ABB RAPID module: P703.mod

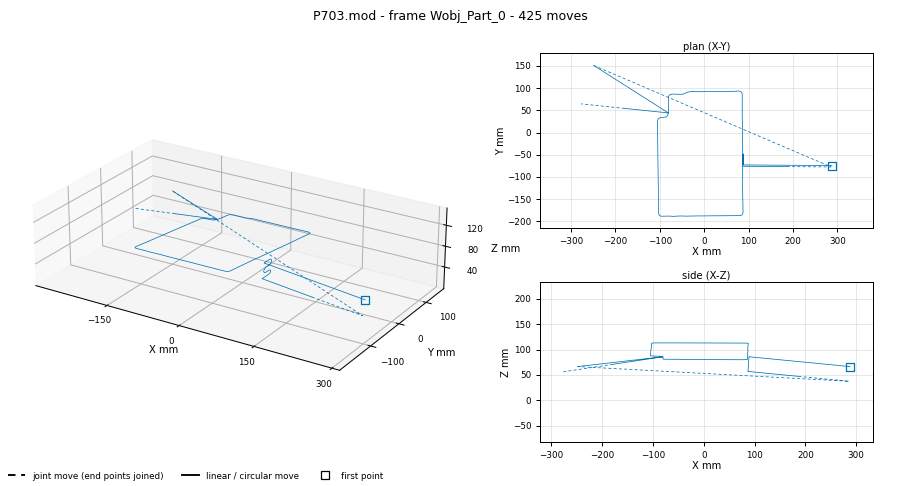
[picture p0: tool path of P703.mod in frame Wobj_Part_0, 425 of 435 moves have a stored position in this frame; points joined in program order, loops and branches not executed]
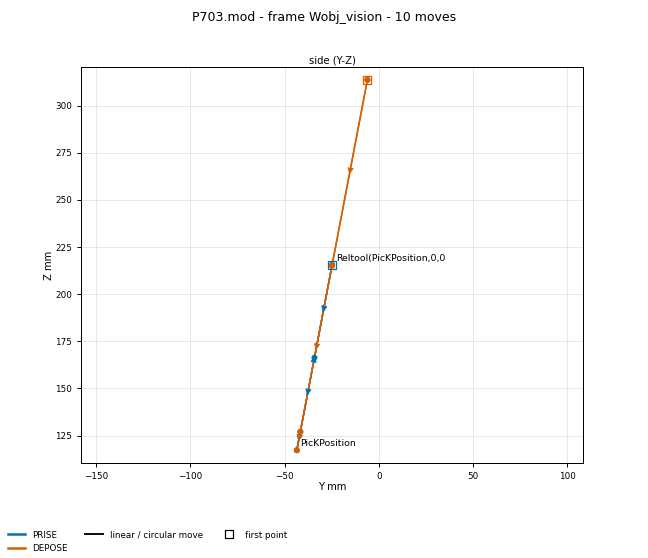
[picture p1: tool path of P703.mod in frame Wobj_vision, 10 of 435 moves have a stored position in this frame; points joined in program order, loops and branches not executed]
MODULE P703

    ! Nom         :P703
    ! Description :
    ! Créé le     :29/05/2023 16:45:30

    LOCAL CONST SPEEDDATA VitesseLente :=[10,500,0,0];
	LOCAL CONST SPEEDDATA VitesseRapide :=[30,500,0,0];
	LOCAL CONST SPEEDDATA VitesseTronconnage :=[2,500,0,0];
	LOCAL CONST SPEEDDATA VitesseTronconnageApp :=[10,500,0,0];
    !
    !Point de prise
    LOCAL PERS Robtarget PicKPosition := [[-18.2045176423154,-43.4890732040902,117.207315713413],[0.0720116404996143,0.704562270319023,0.703344125703762,-0.0609374409822815],[0,0,0,0],[8.999999E+09,8.999999E+09,8.999999E+09,8.999999E+09,8.999999E+09,8.999999E+09]];
	LOCAL PERS Pose Ref := [[0,0,0],[1,0,0,0]];
    !
    !Declaration des points de meulage

    !Tr_meulage_motif_1 : Meulage d'un motif
    LOCAL CONST Robtarget Tr_meulage_motif_1_0 := [[88.8950546875,-72.9881875,85.8599921875],[0.525548833980486,-0.476975326776561,-0.473452006925869,0.521666711498837],[0,0,0,0],[8.999999E+09,8.999999E+09,8.999999E+09,8.999999E+09,8.999999E+09,8.999999E+09]];
    LOCAL CONST Robtarget Tr_meulage_motif_1_1 := [[88.8954296875,-71.9881875,85.8600078125],[0.525548833980486,-0.476975326776561,-0.473452006925869,0.521666711498837],[0,0,0,0],[8.999999E+09,8.999999E+09,8.999999E+09,8.999999E+09,8.999999E+09,8.999999E+09]];
    LOCAL CONST Robtarget Tr_meulage_motif_1_2 := [[88.8958046875,-70.9881875,85.8600234375],[0.525548833980486,-0.476975326776561,-0.473452006925869,0.521666711498837],[0,0,0,0],[8.999999E+09,8.999999E+09,8.999999E+09,8.999999E+09,8.999999E+09,8.999999E+09]];
    LOCAL CONST Robtarget Tr_meulage_motif_1_3 := [[88.8961796875,-69.9881875,85.860046875],[0.525548833980486,-0.476975326776561,-0.473452006925869,0.521666711498837],[0,0,0,0],[8.999999E+09,8.999999E+09,8.999999E+09,8.999999E+09,8.999999E+09,8.999999E+09]];
    LOCAL CONST Robtarget Tr_meulage_motif_1_4 := [[88.8965546875,-68.9881875,85.8600625],[0.525548833980486,-0.476975326776561,-0.473452006925869,0.521666711498837],[0,0,0,0],[8.999999E+09,8.999999E+09,8.999999E+09,8.999999E+09,8.999999E+09,8.999999E+09]];
    LOCAL CONST Robtarget Tr_meulage_motif_1_5 := [[88.8969296875,-67.9881875,85.860078125],[0.525548833980486,-0.476975326776561,-0.473452006925869,0.521666711498837],[0,0,0,0],[8.999999E+09,8.999999E+09,8.999999E+09,8.999999E+09,8.999999E+09,8.999999E+09]];
    LOCAL CONST Robtarget Tr_meulage_motif_1_6 := [[88.8973046875,-66.9881875,85.86009375],[0.525548833980486,-0.476975326776561,-0.473452006925869,0.521666711498837],[0,0,0,0],[8.999999E+09,8.999999E+09,8.999999E+09,8.999999E+09,8.999999E+09,8.999999E+09]];
    LOCAL CONST Robtarget Tr_meulage_motif_1_7 := [[88.897671875,-65.9881875,85.860109375],[0.525548833980486,-0.476975326776561,-0.473452006925869,0.521666711498837],[0,0,0,0],[8.999999E+09,8.999999E+09,8.999999E+09,8.999999E+09,8.999999E+09,8.999999E+09]];
    LOCAL CONST Robtarget Tr_meulage_motif_1_8 := [[88.898046875,-64.98818359375,85.860125],[0.525548833980486,-0.476975326776561,-0.473452006925869,0.521666711498837],[0,0,0,0],[8.999999E+09,8.999999E+09,8.999999E+09,8.999999E+09,8.999999E+09,8.999999E+09]];
    LOCAL CONST Robtarget Tr_meulage_motif_1_9 := [[88.898421875,-63.98818359375,85.8601484375],[0.525548833980486,-0.476975326776561,-0.473452006925869,0.521666711498837],[0,0,0,0],[8.999999E+09,8.999999E+09,8.999999E+09,8.999999E+09,8.999999E+09,8.999999E+09]];
    LOCAL CONST Robtarget Tr_meulage_motif_1_10 := [[88.898796875,-62.98818359375,85.8601640625],[0.525548833980486,-0.476975326776561,-0.473452006925869,0.521666711498837],[0,0,0,0],[8.999999E+09,8.999999E+09,8.999999E+09,8.999999E+09,8.999999E+09,8.999999E+09]];
    LOCAL CONST Robtarget Tr_meulage_motif_1_11 := [[88.899171875,-61.98818359375,85.8601796875],[0.525548833980486,-0.476975326776561,-0.473452006925869,0.521666711498837],[0,0,0,0],[8.999999E+09,8.999999E+09,8.999999E+09,8.999999E+09,8.999999E+09,8.999999E+09]];
    LOCAL CONST Robtarget Tr_meulage_motif_1_12 := [[88.899546875,-60.98818359375,85.8601953125],[0.525548833980486,-0.476975326776561,-0.473452006925869,0.521666711498837],[0,0,0,0],[8.999999E+09,8.999999E+09,8.999999E+09,8.999999E+09,8.999999E+09,8.999999E+09]];
    LOCAL CONST Robtarget Tr_meulage_motif_1_13 := [[88.899921875,-59.98818359375,85.8602109375],[0.525548833980486,-0.476975326776561,-0.473452006925869,0.521666711498837],[0,0,0,0],[8.999999E+09,8.999999E+09,8.999999E+09,8.999999E+09,8.999999E+09,8.999999E+09]];
    LOCAL CONST Robtarget Tr_meulage_motif_1_14 := [[88.900296875,-58.98818359375,85.8602265625],[0.525548833980486,-0.476975326776561,-0.473452006925869,0.521666711498837],[0,0,0,0],[8.999999E+09,8.999999E+09,8.999999E+09,8.999999E+09,8.999999E+09,8.999999E+09]];
    LOCAL CONST Robtarget Tr_meulage_motif_1_15 := [[88.900671875,-57.98818359375,85.8602421875],[0.525548833980486,-0.476975326776561,-0.473452006925869,0.521666711498837],[0,0,0,0],[8.999999E+09,8.999999E+09,8.999999E+09,8.999999E+09,8.999999E+09,8.999999E+09]];
    LOCAL CONST Robtarget Tr_meulage_motif_1_16 := [[88.901046875,-56.98818359375,85.860265625],[0.525548833980486,-0.476975326776561,-0.473452006925869,0.521666711498837],[0,0,0,0],[8.999999E+09,8.999999E+09,8.999999E+09,8.999999E+09,8.999999E+09,8.999999E+09]];
    LOCAL CONST Robtarget Tr_meulage_motif_1_17 := [[88.901421875,-55.98818359375,85.86028125],[0.525548833980486,-0.476975326776561,-0.473452006925869,0.521666711498837],[0,0,0,0],[8.999999E+09,8.999999E+09,8.999999E+09,8.999999E+09,8.999999E+09,8.999999E+09]];
    LOCAL CONST Robtarget Tr_meulage_motif_1_18 := [[88.901796875,-54.98818359375,85.860296875],[0.525548833980486,-0.476975326776561,-0.473452006925869,0.521666711498837],[0,0,0,0],[8.999999E+09,8.999999E+09,8.999999E+09,8.999999E+09,8.999999E+09,8.999999E+09]];
    LOCAL CONST Robtarget Tr_meulage_motif_1_19 := [[88.8946171875,-53.9956171875,85.7499765625],[0.525548833980486,-0.476975326776561,-0.473452006925869,0.521666711498837],[0,0,0,0],[8.999999E+09,8.999999E+09,8.999999E+09,8.999999E+09,8.999999E+09,8.999999E+09]];
    LOCAL CONST Robtarget Tr_meulage_motif_1_20 := [[88.8805546875,-53.049109375,85.539296875],[0.525548833980486,-0.476975326776561,-0.473452006925869,0.521666711498837],[0,0,0,0],[8.999999E+09,8.999999E+09,8.999999E+09,8.999999E+09,8.999999E+09,8.999999E+09]];
    LOCAL CONST Robtarget Tr_meulage_motif_1_21 := [[88.8623203125,-52.19637890625,85.2681015625],[0.525548833980486,-0.476975326776561,-0.473452006925869,0.521666711498837],[0,0,0,0],[8.999999E+09,8.999999E+09,8.999999E+09,8.999999E+09,8.999999E+09,8.999999E+09]];
    LOCAL CONST Robtarget Tr_meulage_motif_1_22 := [[88.843765625,-51.4464296875,84.9928203125],[0.525548833980486,-0.476975326776561,-0.473452006925869,0.521666711498837],[0,0,0,0],[8.999999E+09,8.999999E+09,8.999999E+09,8.999999E+09,8.999999E+09,8.999999E+09]];
    LOCAL CONST Robtarget Tr_meulage_motif_1_23 := [[88.8021171875,-50.34533984375,84.3781484375],[0.525548833980486,-0.476975326776561,-0.473452006925869,0.521666711498837],[0,0,0,0],[8.999999E+09,8.999999E+09,8.999999E+09,8.999999E+09,8.999999E+09,8.999999E+09]];
    LOCAL CONST Robtarget Tr_meulage_motif_1_24 := [[88.744640625,-49.3214296875,83.5324921875],[0.525548833980486,-0.476975326776561,-0.473452006925869,0.521666711498837],[0,0,0,0],[8.999999E+09,8.999999E+09,8.999999E+09,8.999999E+09,8.999999E+09,8.999999E+09]];
    LOCAL CONST Robtarget Tr_meulage_motif_1_25 := [[88.6750625,-48.47373046875,82.511015625],[0.525548833980486,-0.476975326776561,-0.473452006925869,0.521666711498837],[0,0,0,0],[8.999999E+09,8.999999E+09,8.999999E+09,8.999999E+09,8.999999E+09,8.999999E+09]];
    LOCAL CONST Robtarget Tr_meulage_motif_1_26 := [[88.5990546875,-47.98552734375,81.3974453125],[0.525548833980486,-0.476975326776561,-0.473452006925869,0.521666711498837],[0,0,0,0],[8.999999E+09,8.999999E+09,8.999999E+09,8.999999E+09,8.999999E+09,8.999999E+09]];
    LOCAL CONST Robtarget Tr_meulage_motif_1_27 := [[88.5515546875,-47.95843359375,80.70309375],[0.525548833980486,-0.476975326776561,-0.473452006925869,0.521666711498837],[0,0,0,0],[8.999999E+09,8.999999E+09,8.999999E+09,8.999999E+09,8.999999E+09,8.999999E+09]];
    LOCAL CONST Robtarget Tr_meulage_motif_1_28 := [[88.506421875,-47.95840625,80.043390625],[0.525548833980486,-0.476975326776561,-0.473452006925869,0.521666711498837],[0,0,0,0],[8.999999E+09,8.999999E+09,8.999999E+09,8.999999E+09,8.999999E+09,8.999999E+09]];
    LOCAL CONST Robtarget Tr_meulage_motif_1_29 := [[88.4612734375,-48.01325390625,79.3838359375],[0.525548833980486,-0.476975326776561,-0.473452006925869,0.521666711498837],[0,0,0,0],[8.999999E+09,8.999999E+09,8.999999E+09,8.999999E+09,8.999999E+09,8.999999E+09]];
    LOCAL CONST Robtarget Tr_meulage_motif_1_30 := [[88.385875,-48.51142578125,78.2846484375],[0.525548833980486,-0.476975326776561,-0.473452006925869,0.521666711498837],[0,0,0,0],[8.999999E+09,8.999999E+09,8.999999E+09,8.999999E+09,8.999999E+09,8.999999E+09]];
    LOCAL CONST Robtarget Tr_meulage_motif_1_31 := [[88.31684375,-49.3680078125,77.280359375],[0.525548833980486,-0.476975326776561,-0.473452006925869,0.521666711498837],[0,0,0,0],[8.999999E+09,8.999999E+09,8.999999E+09,8.999999E+09,8.999999E+09,8.999999E+09]];
    LOCAL CONST Robtarget Tr_meulage_motif_1_32 := [[88.2598828125,-50.39137890625,76.4533984375],[0.525548833980486,-0.476975326776561,-0.473452006925869,0.521666711498837],[0,0,0,0],[8.999999E+09,8.999999E+09,8.999999E+09,8.999999E+09,8.999999E+09,8.999999E+09]];
    LOCAL CONST Robtarget Tr_meulage_motif_1_33 := [[88.232609375,-51.07845703125,76.0585625],[0.525548833980486,-0.476975326776561,-0.473452006925869,0.521666711498837],[0,0,0,0],[8.999999E+09,8.999999E+09,8.999999E+09,8.999999E+09,8.999999E+09,8.999999E+09]];
    LOCAL CONST Robtarget Tr_meulage_motif_1_34 := [[88.1988984375,-52.23659375,75.5721484375],[0.525548833980486,-0.476975326776561,-0.473452006925869,0.521666711498837],[0,0,0,0],[8.999999E+09,8.999999E+09,8.999999E+09,8.999999E+09,8.999999E+09,8.999999E+09]];
    LOCAL CONST Robtarget Tr_meulage_motif_1_35 := [[88.1805546875,-53.08161328125,75.30865625],[0.525548833980486,-0.476975326776561,-0.473452006925869,0.521666711498837],[0,0,0,0],[8.999999E+09,8.999999E+09,8.999999E+09,8.999999E+09,8.999999E+09,8.999999E+09]];
    LOCAL CONST Robtarget Tr_meulage_motif_1_36 := [[88.16625,-54.0136015625,75.1046484375],[0.525548833980486,-0.476975326776561,-0.473452006925869,0.521666711498837],[0,0,0,0],[8.999999E+09,8.999999E+09,8.999999E+09,8.999999E+09,8.999999E+09,8.999999E+09]];
    LOCAL CONST Robtarget Tr_meulage_motif_1_37 := [[88.15846875,-54.99516015625,74.9962890625],[0.525548833980486,-0.476975326776561,-0.473452006925869,0.521666711498837],[0,0,0,0],[8.999999E+09,8.999999E+09,8.999999E+09,8.999999E+09,8.999999E+09,8.999999E+09]];
    LOCAL CONST Robtarget Tr_meulage_motif_1_38 := [[88.150546875,-55.98771875,74.8859375],[0.525548833980486,-0.476975326776561,-0.473452006925869,0.521666711498837],[0,0,0,0],[8.999999E+09,8.999999E+09,8.999999E+09,8.999999E+09,8.999999E+09,8.999999E+09]];
    LOCAL CONST Robtarget Tr_meulage_motif_1_39 := [[88.150171875,-56.98771875,74.885921875],[0.525548833980486,-0.476975326776561,-0.473452006925869,0.521666711498837],[0,0,0,0],[8.999999E+09,8.999999E+09,8.999999E+09,8.999999E+09,8.999999E+09,8.999999E+09]];
    LOCAL CONST Robtarget Tr_meulage_motif_1_40 := [[88.149796875,-57.98771875,74.88590625],[0.525548833980486,-0.476975326776561,-0.473452006925869,0.521666711498837],[0,0,0,0],[8.999999E+09,8.999999E+09,8.999999E+09,8.999999E+09,8.999999E+09,8.999999E+09]];
    LOCAL CONST Robtarget Tr_meulage_motif_1_41 := [[88.149421875,-58.98771875,74.8858828125],[0.525548833980486,-0.476975326776561,-0.473452006925869,0.521666711498837],[0,0,0,0],[8.999999E+09,8.999999E+09,8.999999E+09,8.999999E+09,8.999999E+09,8.999999E+09]];
    LOCAL CONST Robtarget Tr_meulage_motif_1_42 := [[88.149046875,-59.98771875,74.8858671875],[0.525548833980486,-0.476975326776561,-0.473452006925869,0.521666711498837],[0,0,0,0],[8.999999E+09,8.999999E+09,8.999999E+09,8.999999E+09,8.999999E+09,8.999999E+09]];
    LOCAL CONST Robtarget Tr_meulage_motif_1_43 := [[88.148671875,-60.98771875,74.8858515625],[0.525548833980486,-0.476975326776561,-0.473452006925869,0.521666711498837],[0,0,0,0],[8.999999E+09,8.999999E+09,8.999999E+09,8.999999E+09,8.999999E+09,8.999999E+09]];
    LOCAL CONST Robtarget Tr_meulage_motif_1_44 := [[88.148296875,-61.98771875,74.8858359375],[0.525548833980486,-0.476975326776561,-0.473452006925869,0.521666711498837],[0,0,0,0],[8.999999E+09,8.999999E+09,8.999999E+09,8.999999E+09,8.999999E+09,8.999999E+09]];
    LOCAL CONST Robtarget Tr_meulage_motif_1_45 := [[88.147921875,-62.98771875,74.8858203125],[0.525548833980486,-0.476975326776561,-0.473452006925869,0.521666711498837],[0,0,0,0],[8.999999E+09,8.999999E+09,8.999999E+09,8.999999E+09,8.999999E+09,8.999999E+09]];
    LOCAL CONST Robtarget Tr_meulage_motif_1_46 := [[88.147546875,-63.98771875,74.8858046875],[0.525548833980486,-0.476975326776561,-0.473452006925869,0.521666711498837],[0,0,0,0],[8.999999E+09,8.999999E+09,8.999999E+09,8.999999E+09,8.999999E+09,8.999999E+09]];
    LOCAL CONST Robtarget Tr_meulage_motif_1_47 := [[88.1471796875,-64.98771875,74.8857890625],[0.525548833980486,-0.476975326776561,-0.473452006925869,0.521666711498837],[0,0,0,0],[8.999999E+09,8.999999E+09,8.999999E+09,8.999999E+09,8.999999E+09,8.999999E+09]];
    LOCAL CONST Robtarget Tr_meulage_motif_1_48 := [[88.1468046875,-65.98771875,74.885765625],[0.525548833980486,-0.476975326776561,-0.473452006925869,0.521666711498837],[0,0,0,0],[8.999999E+09,8.999999E+09,8.999999E+09,8.999999E+09,8.999999E+09,8.999999E+09]];
    LOCAL CONST Robtarget Tr_meulage_motif_1_49 := [[88.1388828125,-66.9802734375,74.7754140625],[0.525548833980486,-0.476975326776561,-0.473452006925869,0.521666711498837],[0,0,0,0],[8.999999E+09,8.999999E+09,8.999999E+09,8.999999E+09,8.999999E+09,8.999999E+09]];
    LOCAL CONST Robtarget Tr_meulage_motif_1_50 := [[88.124109375,-67.926765625,74.564703125],[0.525548833980486,-0.476975326776561,-0.473452006925869,0.521666711498837],[0,0,0,0],[8.999999E+09,8.999999E+09,8.999999E+09,8.999999E+09,8.999999E+09,8.999999E+09]];
    LOCAL CONST Robtarget Tr_meulage_motif_1_51 := [[88.105234375,-68.7794765625,74.293484375],[0.525548833980486,-0.476975326776561,-0.473452006925869,0.521666711498837],[0,0,0,0],[8.999999E+09,8.999999E+09,8.999999E+09,8.999999E+09,8.999999E+09,8.999999E+09]];
    LOCAL CONST Robtarget Tr_meulage_motif_1_52 := [[88.084203125,-69.4909609375,73.9900234375],[0.525548833980486,-0.476975326776561,-0.473452006925869,0.521666711498837],[0,0,0,0],[8.999999E+09,8.999999E+09,8.999999E+09,8.999999E+09,8.999999E+09,8.999999E+09]];
    LOCAL CONST Robtarget Tr_meulage_motif_1_53 := [[88.03859375,-70.5253984375,73.329015625],[0.525548833980486,-0.476975326776561,-0.473452006925869,0.521666711498837],[0,0,0,0],[8.999999E+09,8.999999E+09,8.999999E+09,8.999999E+09,8.999999E+09,8.999999E+09]];
    LOCAL CONST Robtarget Tr_meulage_motif_1_54 := [[87.9766875,-71.4273046875,72.429171875],[0.525548833980486,-0.476975326776561,-0.473452006925869,0.521666711498837],[0,0,0,0],[8.999999E+09,8.999999E+09,8.999999E+09,8.999999E+09,8.999999E+09,8.999999E+09]];
    LOCAL CONST Robtarget Tr_meulage_motif_1_55 := [[87.9050859375,-71.9622265625,71.3855703125],[0.525548833980486,-0.476975326776561,-0.473452006925869,0.521666711498837],[0,0,0,0],[8.999999E+09,8.999999E+09,8.999999E+09,8.999999E+09,8.999999E+09,8.999999E+09]];
    LOCAL CONST Robtarget Tr_meulage_motif_1_56 := [[87.8576953125,-72.1469765625,70.6939609375],[0.525548833980486,-0.476975326776561,-0.473452006925869,0.521666711498837],[0,0,0,0],[8.999999E+09,8.999999E+09,8.999999E+09,8.999999E+09,8.999999E+09,8.999999E+09]];
    LOCAL CONST Robtarget Tr_meulage_motif_1_57 := [[87.805109375,-72.2107890625,69.9257578125],[0.525548833980486,-0.476975326776561,-0.473452006925869,0.521666711498837],[0,0,0,0],[8.999999E+09,8.999999E+09,8.999999E+09,8.999999E+09,8.999999E+09,8.999999E+09]];
    LOCAL CONST Robtarget Tr_meulage_motif_1_58 := [[87.7525859375,-72.1438203125,69.1576796875],[0.525548833980486,-0.476975326776561,-0.473452006925869,0.521666711498837],[0,0,0,0],[8.999999E+09,8.999999E+09,8.999999E+09,8.999999E+09,8.999999E+09,8.999999E+09]];
    LOCAL CONST Robtarget Tr_meulage_motif_1_59 := [[87.67709375,-71.7241796875,68.0520234375],[0.525548833980486,-0.476975326776561,-0.473452006925869,0.521666711498837],[0,0,0,0],[8.999999E+09,8.999999E+09,8.999999E+09,8.999999E+09,8.999999E+09,8.999999E+09]];
    LOCAL CONST Robtarget Tr_meulage_motif_1_60 := [[87.637265625,-71.30984375,67.4677109375],[0.525548833980486,-0.476975326776561,-0.473452006925869,0.521666711498837],[0,0,0,0],[8.999999E+09,8.999999E+09,8.999999E+09,8.999999E+09,8.999999E+09,8.999999E+09]];
    LOCAL CONST Robtarget Tr_meulage_motif_1_61 := [[87.5770390625,-70.4226796875,66.582671875],[0.525548833980486,-0.476975326776561,-0.473452006925869,0.521666711498837],[0,0,0,0],[8.999999E+09,8.999999E+09,8.999999E+09,8.999999E+09,8.999999E+09,8.999999E+09]];
    LOCAL CONST Robtarget Tr_meulage_motif_1_62 := [[87.5489765625,-69.8369765625,66.1693359375],[0.525548833980486,-0.476975326776561,-0.473452006925869,0.521666711498837],[0,0,0,0],[8.999999E+09,8.999999E+09,8.999999E+09,8.999999E+09,8.999999E+09,8.999999E+09]];
    LOCAL CONST Robtarget Tr_meulage_motif_1_63 := [[87.5122578125,-68.719046875,65.6265234375],[0.525548833980486,-0.476975326776561,-0.473452006925869,0.521666711498837],[0,0,0,0],[8.999999E+09,8.999999E+09,8.999999E+09,8.999999E+09,8.999999E+09,8.999999E+09]];
    LOCAL CONST Robtarget Tr_meulage_motif_1_64 := [[87.4923984375,-67.8934375,65.33173046875],[0.525548833980486,-0.476975326776561,-0.473452006925869,0.521666711498837],[0,0,0,0],[8.999999E+09,8.999999E+09,8.999999E+09,8.999999E+09,8.999999E+09,8.999999E+09]];
    LOCAL CONST Robtarget Tr_meulage_motif_1_65 := [[87.4787890625,-66.9614296875,65.12775390625],[0.525548833980486,-0.476975326776561,-0.473452006925869,0.521666711498837],[0,0,0,0],[8.999999E+09,8.999999E+09,8.999999E+09,8.999999E+09,8.999999E+09,8.999999E+09]];
    LOCAL CONST Robtarget Tr_meulage_motif_1_66 := [[87.4717421875,-65.979859375,65.0194296875],[0.525548833980486,-0.476975326776561,-0.473452006925869,0.521666711498837],[0,0,0,0],[8.999999E+09,8.999999E+09,8.999999E+09,8.999999E+09,8.999999E+09,8.999999E+09]];
    LOCAL CONST Robtarget Tr_meulage_motif_1_67 := [[87.4645625,-64.98729296875,64.909109375],[0.525548833980486,-0.476975326776561,-0.473452006925869,0.521666711498837],[0,0,0,0],[8.999999E+09,8.999999E+09,8.999999E+09,8.999999E+09,8.999999E+09,8.999999E+09]];
    LOCAL CONST Robtarget Tr_meulage_motif_1_68 := [[87.4649375,-63.98729296875,64.90912890625],[0.525548833980486,-0.476975326776561,-0.473452006925869,0.521666711498837],[0,0,0,0],[8.999999E+09,8.999999E+09,8.999999E+09,8.999999E+09,8.999999E+09,8.999999E+09]];
    LOCAL CONST Robtarget Tr_meulage_motif_1_69 := [[87.4653125,-62.98729296875,64.90914453125],[0.525548833980486,-0.476975326776561,-0.473452006925869,0.521666711498837],[0,0,0,0],[8.999999E+09,8.999999E+09,8.999999E+09,8.999999E+09,8.999999E+09,8.999999E+09]];
    LOCAL CONST Robtarget Tr_meulage_motif_1_70 := [[87.4656875,-61.987296875,64.90916015625],[0.525548833980486,-0.476975326776561,-0.473452006925869,0.521666711498837],[0,0,0,0],[8.999999E+09,8.999999E+09,8.999999E+09,8.999999E+09,8.999999E+09,8.999999E+09]];
    LOCAL CONST Robtarget Tr_meulage_motif_1_71 := [[87.4660625,-60.987296875,64.9091796875],[0.525548833980486,-0.476975326776561,-0.473452006925869,0.521666711498837],[0,0,0,0],[8.999999E+09,8.999999E+09,8.999999E+09,8.999999E+09,8.999999E+09,8.999999E+09]];
    LOCAL CONST Robtarget Tr_meulage_motif_1_72 := [[87.4664375,-59.987296875,64.9091953125],[0.525548833980486,-0.476975326776561,-0.473452006925869,0.521666711498837],[0,0,0,0],[8.999999E+09,8.999999E+09,8.999999E+09,8.999999E+09,8.999999E+09,8.999999E+09]];
    LOCAL CONST Robtarget Tr_meulage_motif_1_73 := [[87.4668125,-58.987296875,64.9092109375],[0.525548833980486,-0.476975326776561,-0.473452006925869,0.521666711498837],[0,0,0,0],[8.999999E+09,8.999999E+09,8.999999E+09,8.999999E+09,8.999999E+09,8.999999E+09]];
    LOCAL CONST Robtarget Tr_meulage_motif_1_74 := [[87.4671875,-57.987296875,64.90923046875],[0.525548833980486,-0.476975326776561,-0.473452006925869,0.521666711498837],[0,0,0,0],[8.999999E+09,8.999999E+09,8.999999E+09,8.999999E+09,8.999999E+09,8.999999E+09]];
    LOCAL CONST Robtarget Tr_meulage_motif_1_75 := [[87.4675625,-56.987296875,64.90924609375],[0.525548833980486,-0.476975326776561,-0.473452006925869,0.521666711498837],[0,0,0,0],[8.999999E+09,8.999999E+09,8.999999E+09,8.999999E+09,8.999999E+09,8.999999E+09]];
    LOCAL CONST Robtarget Tr_meulage_motif_1_76 := [[87.4679296875,-55.987296875,64.90926171875],[0.525548833980486,-0.476975326776561,-0.473452006925869,0.521666711498837],[0,0,0,0],[8.999999E+09,8.999999E+09,8.999999E+09,8.999999E+09,8.999999E+09,8.999999E+09]];
    LOCAL CONST Robtarget Tr_meulage_motif_1_77 := [[87.4683046875,-54.987296875,64.90927734375],[0.525548833980486,-0.476975326776561,-0.473452006925869,0.521666711498837],[0,0,0,0],[8.999999E+09,8.999999E+09,8.999999E+09,8.999999E+09,8.999999E+09,8.999999E+09]];
    LOCAL CONST Robtarget Tr_meulage_motif_1_78 := [[87.4611328125,-53.9947265625,64.7989609375],[0.525548833980486,-0.476975326776561,-0.473452006925869,0.521666711498837],[0,0,0,0],[8.999999E+09,8.999999E+09,8.999999E+09,8.999999E+09,8.999999E+09,8.999999E+09]];
    LOCAL CONST Robtarget Tr_meulage_motif_1_79 := [[87.4470703125,-53.04821875,64.58828125],[0.525548833980486,-0.476975326776561,-0.473452006925869,0.521666711498837],[0,0,0,0],[8.999999E+09,8.999999E+09,8.999999E+09,8.999999E+09,8.999999E+09,8.999999E+09]];
    LOCAL CONST Robtarget Tr_meulage_motif_1_80 := [[87.428828125,-52.19548828125,64.3170859375],[0.525548833980486,-0.476975326776561,-0.473452006925869,0.521666711498837],[0,0,0,0],[8.999999E+09,8.999999E+09,8.999999E+09,8.999999E+09,8.999999E+09,8.999999E+09]];
    LOCAL CONST Robtarget Tr_meulage_motif_1_81 := [[87.4102734375,-51.4455390625,64.0418046875],[0.525548833980486,-0.476975326776561,-0.473452006925869,0.521666711498837],[0,0,0,0],[8.999999E+09,8.999999E+09,8.999999E+09,8.999999E+09,8.999999E+09,8.999999E+09]];
    LOCAL CONST Robtarget Tr_meulage_motif_1_82 := [[87.3686328125,-50.344453125,63.42713671875],[0.525548833980486,-0.476975326776561,-0.473452006925869,0.521666711498837],[0,0,0,0],[8.999999E+09,8.999999E+09,8.999999E+09,8.999999E+09,8.999999E+09,8.999999E+09]];
    LOCAL CONST Robtarget Tr_meulage_motif_1_83 := [[87.30796875,-49.3876953125,62.53526953125],[0.525548833980486,-0.476975326776561,-0.473452006925869,0.521666711498837],[0,0,0,0],[8.999999E+09,8.999999E+09,8.999999E+09,8.999999E+09,8.999999E+09,8.999999E+09]];
    LOCAL CONST Robtarget Tr_meulage_motif_1_84 := [[87.2340625,-48.7785234375,61.4518125],[0.525548833980486,-0.476975326776561,-0.473452006925869,0.521666711498837],[0,0,0,0],[8.999999E+09,8.999999E+09,8.999999E+09,8.999999E+09,8.999999E+09,8.999999E+09]];
    LOCAL CONST Robtarget Tr_meulage_motif_1_85 := [[87.1669296875,-48.60916796875,60.469734375],[0.525548833980486,-0.476975326776561,-0.473452006925869,0.521666711498837],[0,0,0,0],[8.999999E+09,8.999999E+09,8.999999E+09,8.999999E+09,8.999999E+09,8.999999E+09]];
    LOCAL CONST Robtarget Tr_meulage_motif_1_86 := [[87.1529140625,-48.74062890625,60.2655546875],[0.525548833980486,-0.476975326776561,-0.473452006925869,0.521666711498837],[0,0,0,0],[8.999999E+09,8.999999E+09,8.999999E+09,8.999999E+09,8.999999E+09,8.999999E+09]];
    LOCAL CONST Robtarget Tr_meulage_motif_1_87 := [[87.10328125,-48.86397265625,59.54083984375],[0.525548833980486,-0.476975326776561,-0.473452006925869,0.521666711498837],[0,0,0,0],[8.999999E+09,8.999999E+09,8.999999E+09,8.999999E+09,8.999999E+09,8.999999E+09]];
    LOCAL CONST Robtarget Tr_meulage_motif_1_88 := [[87.0390703125,-49.54793359375,58.606109375],[0.525548833980486,-0.476975326776561,-0.473452006925869,0.521666711498837],[0,0,0,0],[8.999999E+09,8.999999E+09,8.999999E+09,8.999999E+09,8.999999E+09,8.999999E+09]];
    LOCAL CONST Robtarget Tr_meulage_motif_1_89 := [[87.007203125,-50.1055390625,58.1433671875],[0.525548833980486,-0.476975326776561,-0.473452006925869,0.521666711498837],[0,0,0,0],[8.999999E+09,8.999999E+09,8.999999E+09,8.999999E+09,8.999999E+09,8.999999E+09]];
    LOCAL CONST Robtarget Tr_meulage_motif_1_90 := [[86.9705703125,-51.235828125,57.6141484375],[0.525548833980486,-0.476975326776561,-0.473452006925869,0.521666711498837],[0,0,0,0],[8.999999E+09,8.999999E+09,8.999999E+09,8.999999E+09,8.999999E+09,8.999999E+09]];
    LOCAL CONST Robtarget Tr_meulage_motif_1_91 := [[86.9522265625,-52.0808515625,57.35065625],[0.525548833980486,-0.476975326776561,-0.473452006925869,0.521666711498837],[0,0,0,0],[8.999999E+09,8.999999E+09,8.999999E+09,8.999999E+09,8.999999E+09,8.999999E+09]];
    LOCAL CONST Robtarget Tr_meulage_motif_1_92 := [[86.937921875,-53.01283984375,57.1466484375],[0.525548833980486,-0.476975326776561,-0.473452006925869,0.521666711498837],[0,0,0,0],[8.999999E+09,8.999999E+09,8.999999E+09,8.999999E+09,8.999999E+09,8.999999E+09]];
    LOCAL CONST Robtarget Tr_meulage_motif_1_93 := [[86.930140625,-53.9943984375,57.03829296875],[0.525548833980486,-0.476975326776561,-0.473452006925869,0.521666711498837],[0,0,0,0],[8.999999E+09,8.999999E+09,8.999999E+09,8.999999E+09,8.999999E+09,8.999999E+09]];
    LOCAL CONST Robtarget Tr_meulage_motif_1_94 := [[86.92221875,-54.98695703125,56.9279375],[0.525548833980486,-0.476975326776561,-0.473452006925869,0.521666711498837],[0,0,0,0],[8.999999E+09,8.999999E+09,8.999999E+09,8.999999E+09,8.999999E+09,8.999999E+09]];
    LOCAL CONST Robtarget Tr_meulage_motif_1_95 := [[86.92184375,-55.98695703125,56.927921875],[0.525548833980486,-0.476975326776561,-0.473452006925869,0.521666711498837],[0,0,0,0],[8.999999E+09,8.999999E+09,8.999999E+09,8.999999E+09,8.999999E+09,8.999999E+09]];
    LOCAL CONST Robtarget Tr_meulage_motif_1_96 := [[86.92146875,-56.98695703125,56.92790625],[0.525548833980486,-0.476975326776561,-0.473452006925869,0.521666711498837],[0,0,0,0],[8.999999E+09,8.999999E+09,8.999999E+09,8.999999E+09,8.999999E+09,8.999999E+09]];
    LOCAL CONST Robtarget Tr_meulage_motif_1_97 := [[86.92109375,-57.98695703125,56.92788671875],[0.525548833980486,-0.476975326776561,-0.473452006925869,0.521666711498837],[0,0,0,0],[8.999999E+09,8.999999E+09,8.999999E+09,8.999999E+09,8.999999E+09,8.999999E+09]];
    LOCAL CONST Robtarget Tr_meulage_motif_1_98 := [[86.92071875,-58.98695703125,56.92787109375],[0.525548833980486,-0.476975326776561,-0.473452006925869,0.521666711498837],[0,0,0,0],[8.999999E+09,8.999999E+09,8.999999E+09,8.999999E+09,8.999999E+09,8.999999E+09]];
    LOCAL CONST Robtarget Tr_meulage_motif_1_99 := [[86.92034375,-59.98695703125,56.92785546875],[0.525548833980486,-0.476975326776561,-0.473452006925869,0.521666711498837],[0,0,0,0],[8.999999E+09,8.999999E+09,8.999999E+09,8.999999E+09,8.999999E+09,8.999999E+09]];
    LOCAL CONST Robtarget Tr_meulage_motif_1_100 := [[86.91996875,-60.98695703125,56.92783984375],[0.525548833980486,-0.476975326776561,-0.473452006925869,0.521666711498837],[0,0,0,0],[8.999999E+09,8.999999E+09,8.999999E+09,8.999999E+09,8.999999E+09,8.999999E+09]];
    LOCAL CONST Robtarget Tr_meulage_motif_1_101 := [[86.91959375,-61.98695703125,56.9278203125],[0.525548833980486,-0.476975326776561,-0.473452006925869,0.521666711498837],[0,0,0,0],[8.999999E+09,8.999999E+09,8.999999E+09,8.999999E+09,8.999999E+09,8.999999E+09]];
    LOCAL CONST Robtarget Tr_meulage_motif_1_102 := [[86.9192265625,-62.98695703125,56.9278046875],[0.525548833980486,-0.476975326776561,-0.473452006925869,0.521666711498837],[0,0,0,0],[8.999999E+09,8.999999E+09,8.999999E+09,8.999999E+09,8.999999E+09,8.999999E+09]];
    LOCAL CONST Robtarget Tr_meulage_motif_1_103 := [[86.9188515625,-63.98695703125,56.9277890625],[0.525548833980486,-0.476975326776561,-0.473452006925869,0.521666711498837],[0,0,0,0],[8.999999E+09,8.999999E+09,8.999999E+09,8.999999E+09,8.999999E+09,8.999999E+09]];
    LOCAL CONST Robtarget Tr_meulage_motif_1_104 := [[86.9184765625,-64.98695703125,56.92776953125],[0.525548833980486,-0.476975326776561,-0.473452006925869,0.521666711498837],[0,0,0,0],[8.999999E+09,8.999999E+09,8.999999E+09,8.999999E+09,8.999999E+09,8.999999E+09]];
    LOCAL CONST Robtarget Tr_meulage_motif_1_105 := [[86.9181015625,-65.986953125,56.92775390625],[0.525548833980486,-0.476975326776561,-0.473452006925869,0.521666711498837],[0,0,0,0],[8.999999E+09,8.999999E+09,8.999999E+09,8.999999E+09,8.999999E+09,8.999999E+09]];
    LOCAL CONST Robtarget Tr_meulage_motif_1_106 := [[86.9177265625,-66.986953125,56.92773828125],[0.525548833980486,-0.476975326776561,-0.473452006925869,0.521666711498837],[0,0,0,0],[8.999999E+09,8.999999E+09,8.999999E+09,8.999999E+09,8.999999E+09,8.999999E+09]];
    LOCAL CONST Robtarget Tr_meulage_motif_1_107 := [[86.9173515625,-67.986953125,56.92771875],[0.525548833980486,-0.476975326776561,-0.473452006925869,0.521666711498837],[0,0,0,0],[8.999999E+09,8.999999E+09,8.999999E+09,8.999999E+09,8.999999E+09,8.999999E+09]];
    LOCAL CONST Robtarget Tr_meulage_motif_1_108 := [[86.9169765625,-68.986953125,56.927703125],[0.525548833980486,-0.476975326776561,-0.473452006925869,0.521666711498837],[0,0,0,0],[8.999999E+09,8.999999E+09,8.999999E+09,8.999999E+09,8.999999E+09,8.999999E+09]];
    LOCAL CONST Robtarget Tr_meulage_motif_1_109 := [[86.9166015625,-69.986953125,56.9276875],[0.525548833980486,-0.476975326776561,-0.473452006925869,0.521666711498837],[0,0,0,0],[8.999999E+09,8.999999E+09,8.999999E+09,8.999999E+09,8.999999E+09,8.999999E+09]];
    LOCAL CONST Robtarget Tr_meulage_motif_1_110 := [[86.9162265625,-70.986953125,56.92766796875],[0.525548833980486,-0.476975326776561,-0.473452006925869,0.521666711498837],[0,0,0,0],[8.999999E+09,8.999999E+09,8.999999E+09,8.999999E+09,8.999999E+09,8.999999E+09]];
    LOCAL CONST Robtarget Tr_meulage_motif_1_111 := [[86.9158515625,-71.986953125,56.92765234375],[0.525548833980486,-0.476975326776561,-0.473452006925869,0.521666711498837],[0,0,0,0],[8.999999E+09,8.999999E+09,8.999999E+09,8.999999E+09,8.999999E+09,8.999999E+09]];
    LOCAL CONST Robtarget Tr_meulage_motif_1_112 := [[86.9154765625,-72.986953125,56.92763671875],[0.525548833980486,-0.476975326776561,-0.473452006925869,0.521666711498837],[0,0,0,0],[8.999999E+09,8.999999E+09,8.999999E+09,8.999999E+09,8.999999E+09,8.999999E+09]];
    LOCAL CONST Robtarget Tr_meulage_motif_1_113 := [[86.9151015625,-73.986953125,56.9276171875],[0.525548833980486,-0.476975326776561,-0.473452006925869,0.521666711498837],[0,0,0,0],[8.999999E+09,8.999999E+09,8.999999E+09,8.999999E+09,8.999999E+09,8.999999E+09]];
    LOCAL CONST Robtarget Tr_meulage_motif_1_114 := [[86.914734375,-74.986953125,56.9276015625],[0.525548833980486,-0.476975326776561,-0.473452006925869,0.521666711498837],[0,0,0,0],[8.999999E+09,8.999999E+09,8.999999E+09,8.999999E+09,8.999999E+09,8.999999E+09]];
    LOCAL CONST Robtarget Tr_meulage_motif_1_115 := [[86.914359375,-75.986953125,56.9275859375],[0.525548833980486,-0.476975326776561,-0.473452006925869,0.521666711498837],[0,0,0,0],[8.999999E+09,8.999999E+09,8.999999E+09,8.999999E+09,8.999999E+09,8.999999E+09]];

    !Tr_meulage_bavure : Meulage de la bavure
    LOCAL CONST Robtarget Tr_meulage_bavure_0 := [[-80.6398046875,44.21337109375,85.806125],[0.356467501522501,-0.323594070063004,0.589118545755795,-0.648966206535397],[0,0,0,0],[8.999999E+09,8.999999E+09,8.999999E+09,8.999999E+09,8.999999E+09,8.999999E+09]];
    LOCAL CONST Robtarget Tr_meulage_bavure_1 := [[-80.89575,42.674421875,85.98690625],[0.352265354142538,-0.319790237292867,0.59120614434461,-0.651243901539342],[0,0,0,0],[8.999999E+09,8.999999E+09,8.999999E+09,8.999999E+09,8.999999E+09,8.999999E+09]];
    LOCAL CONST Robtarget Tr_meulage_bavure_2 := [[-81.150265625,42.21675390625,86.040671875],[0.339738788803568,-0.308447042706282,0.597240975604926,-0.657830672959623],[0,0,0,0],[8.999999E+09,8.999999E+09,8.999999E+09,8.999999E+09,8.999999E+09,8.999999E+09]];
    LOCAL CONST Robtarget Tr_meulage_bavure_3 := [[-81.6705,41.09446484375,86.1725078125],[0.31931681091922,-0.289948319035797,0.606496970705713,-0.667928267913171],[0,0,0,0],[8.999999E+09,8.999999E+09,8.999999E+09,8.999999E+09,8.999999E+09,8.999999E+09]];
    LOCAL CONST Robtarget Tr_meulage_bavure_4 := [[-81.9177890625,39.7865625,86.32615625],[0.292123359571493,-0.265311215268551,0.617755456543852,-0.680185340738601],[0,0,0,0],[8.999999E+09,8.999999E+09,8.999999E+09,8.999999E+09,8.999999E+09,8.999999E+09]];
    LOCAL CONST Robtarget Tr_meulage_bavure_5 := [[-82.8616015625,38.1317734375,86.520546875],[0.260439952462833,-0.236595524688921,0.629411963893967,-0.692844981626821],[0,0,0,0],[8.999999E+09,8.999999E+09,8.999999E+09,8.999999E+09,8.999999E+09,8.999999E+09]];
    LOCAL CONST Robtarget Tr_meulage_bavure_6 := [[-83.6377578125,36.96069140625,86.6581171875],[0.227630067036962,-0.206856749254602,0.639928253768548,-0.704192209483536],[0,0,0,0],[8.999999E+09,8.999999E+09,8.999999E+09,8.999999E+09,8.999999E+09,8.999999E+09]];
    LOCAL CONST Robtarget Tr_meulage_bavure_7 := [[-85.3959375,35.49608984375,86.8301640625],[0.197468494762164,-0.179516488836576,0.648275884275376,-0.713104762064546],[0,0,0,0],[8.999999E+09,8.999999E+09,8.999999E+09,8.999999E+09,8.999999E+09,8.999999E+09]];
    LOCAL CONST Robtarget Tr_meulage_bavure_8 := [[-85.78003125,34.79388671875,86.91265625],[0.173339170461957,-0.157647449871022,0.654098365680512,-0.719205215183265],[0,0,0,0],[8.999999E+09,8.999999E+09,8.999999E+09,8.999999E+09,8.999999E+09,8.999999E+09]];
    LOCAL CONST Robtarget Tr_meulage_bavure_9 := [[-86.516359375,34.9561328125,86.8936015625],[0.157530751227302,-0.143341765061926,0.657570016377366,-0.722660967790681],[0,0,0,0],[8.999999E+09,8.999999E+09,8.999999E+09,8.999999E+09,8.999999E+09,8.999999E+09]];
    LOCAL CONST Robtarget Tr_meulage_bavure_10 := [[-87.2612890625,34.8977265625,86.9004609375],[0.151203909152679,-0.137660267428464,0.658989108837979,-0.723823447438253],[0,0,0,0],[8.999999E+09,8.999999E+09,8.999999E+09,8.999999E+09,8.999999E+09,8.999999E+09]];
    LOCAL CONST Robtarget Tr_meulage_bavure_11 := [[-93.1481953125,34.1341484375,86.99015625],[0.154618031247686,-0.140851403522588,0.658535812377187,-0.722900221576619],[0,0,0,0],[8.999999E+09,8.999999E+09,8.999999E+09,8.999999E+09,8.999999E+09,8.999999E+09]];
    LOCAL CONST Robtarget Tr_meulage_bavure_12 := [[-93.7944609375,34.12390234375,86.991359375],[0.167469129678402,-0.152656809829176,0.656143627058399,-0.719809370380927],[0,0,0,0],[8.999999E+09,8.999999E+09,8.999999E+09,8.999999E+09,8.999999E+09,8.999999E+09]];
    LOCAL CONST Robtarget Tr_meulage_bavure_13 := [[-96.642515625,33.70594140625,87.0404609375],[0.188962386880001,-0.172369961838228,0.651509863069908,-0.714224552170485],[0,0,0,0],[8.999999E+09,8.999999E+09,8.999999E+09,8.999999E+09,8.999999E+09,8.999999E+09]];
    LOCAL CONST Robtarget Tr_meulage_bavure_14 := [[-97.4105546875,33.61913671875,87.05065625],[0.217772248870419,-0.198801072239124,0.644229278409411,-0.705706750809842],[0,0,0,0],[8.999999E+09,8.999999E+09,8.999999E+09,8.999999E+09,8.999999E+09,8.999999E+09]];
    LOCAL CONST Robtarget Tr_meulage_bavure_15 := [[-100.112515625,32.99455859375,87.12403125],[0.251974945105935,-0.230207504861465,0.633997430009606,-0.693945524148355],[0,0,0,0],[8.999999E+09,8.999999E+09,8.999999E+09,8.999999E+09,8.999999E+09,8.999999E+09]];
    LOCAL CONST Robtarget Tr_meulage_bavure_16 := [[-101.1128203125,32.57331640625,87.173515625],[0.289115969271583,-0.264361107262769,0.620867468778267,-0.679005705051013],[0,0,0,0],[8.999999E+09,8.999999E+09,8.999999E+09,8.999999E+09,8.999999E+09,8.999999E+09]];
    LOCAL CONST Robtarget Tr_meulage_bavure_17 := [[-103.1066875,31.09847265625,87.346765625],[0.326648729588831,-0.298946924277265,0.605340155819241,-0.661433775729591],[0,0,0,0],[8.999999E+09,8.999999E+09,8.999999E+09,8.999999E+09,8.999999E+09,8.999999E+09]];
    LOCAL CONST Robtarget Tr_meulage_bavure_18 := [[-103.8987734375,29.99140234375,87.4768203125],[0.36228718822458,-0.33187058320784,0.588326343444787,-0.642247633595097],[0,0,0,0],[8.999999E+09,8.999999E+09,8.999999E+09,8.999999E+09,8.999999E+09,8.999999E+09]];
    LOCAL CONST Robtarget Tr_meulage_bavure_19 := [[-104.4775390625,28.618578125,87.6380859375],[0.394458747313302,-0.361688409511382,0.570897687828291,-0.622623177472103],[0,0,0,0],[8.999999E+09,8.999999E+09,8.999999E+09,8.999999E+09,8.999999E+09,8.999999E+09]];
    LOCAL CONST Robtarget Tr_meulage_bavure_20 := [[-105.0432421875,26.694552734375,87.864109375],[0.422328884039895,-0.387641863144865,0.554064214099537,-0.603643061997285],[0,0,0,0],[8.999999E+09,8.999999E+09,8.999999E+09,8.999999E+09,8.999999E+09,8.999999E+09]];
    LOCAL CONST Robtarget Tr_meulage_bavure_21 := [[-105.086734375,26.120861328125,87.9315078125],[0.445678795067052,-0.409507690428794,0.538593373947137,-0.58616639331123],[0,0,0,0],[8.999999E+09,8.999999E+09,8.999999E+09,8.999999E+09,8.999999E+09,8.999999E+09]];
    LOCAL CONST Robtarget Tr_meulage_bavure_22 := [[-105.090328125,22.444509765625,88.363375],[0.464743064643507,-0.427484468322051,0.524948233700071,-0.570701555232111],[0,0,0,0],[8.999999E+09,8.999999E+09,8.999999E+09,8.999999E+09,8.999999E+09,8.999999E+09]];
    LOCAL CONST Robtarget Tr_meulage_bavure_23 := [[-105.0225234375,17.2730390625,88.9708828125],[0.479961436932852,-0.441976413867208,0.513347239490675,-0.557466124845033],[0,0,0,0],[8.999999E+09,8.999999E+09,8.999999E+09,8.999999E+09,8.999999E+09,8.999999E+09]];
    LOCAL CONST Robtarget Tr_meulage_bavure_24 := [[-105.0301796875,16.856533203125,89.0198125],[0.491867374238999,-0.45346391768078,0.503798642494302,-0.546464902204825],[0,0,0,0],[8.999999E+09,8.999999E+09,8.999999E+09,8.999999E+09,8.999999E+09,8.999999E+09]];
    LOCAL CONST Robtarget Tr_meulage_bavure_25 := [[-105.0289921875,15.9423173828125,89.1272109375],[0.50098186557085,-0.462412497742938,0.496189356038023,-0.537576018117308],[0,0,0,0],[8.999999E+09,8.999999E+09,8.999999E+09,8.999999E+09,8.999999E+09,8.999999E+09]];
    LOCAL CONST Robtarget Tr_meulage_bavure_26 := [[-104.9676796875,11.2968310546875,89.6729296875],[0.507796100564899,-0.469271824835869,0.490323059752891,-0.530575509933186],[0,0,0,0],[8.999999E+09,8.999999E+09,8.999999E+09,8.999999E+09,8.999999E+09,8.999999E+09]];
    LOCAL CONST Robtarget Tr_meulage_bavure_27 := [[-104.8709375,5.9843017578125,90.2970078125],[0.512747165231321,-0.474436815395772,0.485963327841786,-0.525204433280317],[0,0,0,0],[8.999999E+09,8.999999E+09,8.999999E+09,8.999999E+09,8.999999E+09,8.999999E+09]];
    LOCAL CONST Robtarget Tr_meulage_bavure_28 := [[-104.8862890625,1.80897204589844,90.7874921875],[0.516232265972859,-0.478265191154658,0.482846583012533,-0.521177351552661],[0,0,0,0],[8.999999E+09,8.999999E+09,8.999999E+09,8.999999E+09,8.999999E+09,8.999999E+09]];
    LOCAL CONST Robtarget Tr_meulage_bavure_29 := [[-104.8908671875,1.23067321777344,90.8554296875],[0.518580680708764,-0.481059252614234,0.480728467876961,-0.518224095582731],[0,0,0,0],[8.999999E+09,8.999999E+09,8.999999E+09,8.999999E+09,8.999999E+09,8.999999E+09]];
    LOCAL CONST Robtarget Tr_meulage_bavure_30 := [[-104.8864765625,0.628551391601562,90.9261640625],[0.52005500886692,-0.483062948140571,0.479398780025659,-0.516110245583323],[0,0,0,0],[8.999999E+09,8.999999E+09,8.999999E+09,8.999999E+09,8.999999E+09,8.999999E+09]];
    LOCAL CONST Robtarget Tr_meulage_bavure_31 := [[-104.8773828125,-0.455304229736328,91.053484375],[0.520886921688218,-0.484484627061152,0.478658803272869,-0.51462336811009],[0,0,0,0],[8.999999E+09,8.999999E+09,8.999999E+09,8.999999E+09,8.999999E+09,8.999999E+09]];
    LOCAL CONST Robtarget Tr_meulage_bavure_32 := [[-104.865359375,-4.46175146484375,91.5241328125],[0.521236299775067,-0.485471444253093,0.478367753020309,-0.513609277059822],[0,0,0,0],[8.999999E+09,8.999999E+09,8.999999E+09,8.999999E+09,8.999999E+09,8.999999E+09]];
    LOCAL CONST Robtarget Tr_meulage_bavure_33 := [[-104.8167734375,-5.79502099609375,91.6807578125],[0.521243242385645,-0.486143568126117,0.47839771859772,-0.512938140790295],[0,0,0,0],[8.999999E+09,8.999999E+09,8.999999E+09,8.999999E+09,8.999999E+09,8.999999E+09]];
    LOCAL CONST Robtarget Tr_meulage_bavure_34 := [[-104.7633671875,-9.5107431640625,92.1172578125],[0.520987005477858,-0.486587225744244,0.478676753757433,-0.512517294613538],[0,0,0,0],[8.999999E+09,8.999999E+09,8.999999E+09,8.999999E+09,8.999999E+09,8.999999E+09]];
    LOCAL CONST Robtarget Tr_meulage_bavure_35 := [[-104.6730078125,-12.3688662109375,92.4530078125],[0.520537362215524,-0.486852394491846,0.479139041207859,-0.512290327554282],[0,0,0,0],[8.999999E+09,8.999999E+09,8.999999E+09,8.999999E+09,8.999999E+09,8.999999E+09]];
    LOCAL CONST Robtarget Tr_meulage_bavure_36 := [[-104.7241484375,-13.9786162109375,92.642109375],[0.519957184020112,-0.48700294063968,0.479725636101377,-0.512187442896942],[0,0,0,0],[8.999999E+09,8.999999E+09,8.999999E+09,8.999999E+09,8.999999E+09,8.999999E+09]];
    LOCAL CONST Robtarget Tr_meulage_bavure_37 := [[-104.7202421875,-15.5373251953125,92.82521875],[0.519288186245677,-0.48708278176929,0.480397313757308,-0.51216068207578],[0,0,0,0],[8.999999E+09,8.999999E+09,8.999999E+09,8.999999E+09,8.999999E+09,8.999999E+09]];
    LOCAL CONST Robtarget Tr_meulage_bavure_38 := [[-104.5984765625,-19.052248046875,93.238125],[0.51858313749804,-0.48713763883378,0.481103760149521,-0.512159762480547],[0,0,0,0],[8.999999E+09,8.999999E+09,8.999999E+09,8.999999E+09,8.999999E+09,8.999999E+09]];
    LOCAL CONST Robtarget Tr_meulage_bavure_39 := [[-104.5743125,-19.835771484375,93.3301640625],[0.517880485091653,-0.487193309468091,0.481807901814784,-0.51215586311161],[0,0,0,0],[8.999999E+09,8.999999E+09,8.999999E+09,8.999999E+09,8.999999E+09,8.999999E+09]];
    LOCAL CONST Robtarget Tr_meulage_bavure_40 := [[-104.6134921875,-24.584943359375,93.8880703125],[0.517205126209082,-0.487288338760395,0.482486798727777,-0.512108798386245],[0,0,0,0],[8.999999E+09,8.999999E+09,8.999999E+09,8.999999E+09,8.999999E+09,8.999999E+09]];
    LOCAL CONST Robtarget Tr_meulage_bavure_41 := [[-104.6064765625,-25.341369140625,93.9769296875],[0.516600131610275,-0.487450682348673,0.483098783331736,-0.511987989938687],[0,0,0,0],[8.999999E+09,8.999999E+09,8.999999E+09,8.999999E+09,8.999999E+09,8.999999E+09]];
    LOCAL CONST Robtarget Tr_meulage_bavure_42 := [[-104.603640625,-26.121982421875,94.068625],[0.516075677568263,-0.487703321766225,0.483634670034338,-0.511770330227755],[0,0,0,0],[8.999999E+09,8.999999E+09,8.999999E+09,8.999999E+09,8.999999E+09,8.999999E+09]];
    LOCAL CONST Robtarget Tr_meulage_bavure_43 := [[-104.560546875,-30.81462890625,94.619890625],[0.515636503077161,-0.488048581596106,0.484089559858848,-0.511453689723764],[0,0,0,0],[8.999999E+09,8.999999E+09,8.999999E+09,8.999999E+09,8.999999E+09,8.999999E+09]];
    LOCAL CONST Robtarget Tr_meulage_bavure_44 := [[-104.5008203125,-36.210328125,95.253734375],[0.515276488371758,-0.488471723763139,0.48446850859818,-0.511053597768172],[0,0,0,0],[8.999999E+09,8.999999E+09,8.999999E+09,8.999999E+09,8.999999E+09,8.999999E+09]];
    LOCAL CONST Robtarget Tr_meulage_bavure_45 := [[-104.5387265625,-38.3719453125,95.5076640625],[0.514973172796702,-0.488957246767082,0.484792871873926,-0.510587224197673],[0,0,0,0],[8.999999E+09,8.999999E+09,8.999999E+09,8.999999E+09,8.999999E+09,8.999999E+09]];
    LOCAL CONST Robtarget Tr_meulage_bavure_46 := [[-104.5440078125,-41.5642578125,95.8826796875],[0.514705308141592,-0.489487066940944,0.485082756661742,-0.510074088988909],[0,0,0,0],[8.999999E+09,8.999999E+09,8.999999E+09,8.999999E+09,8.999999E+09,8.999999E+09]];
    LOCAL CONST Robtarget Tr_meulage_bavure_47 := [[-104.4025546875,-45.928109375,96.3953125],[0.514453211866767,-0.490043218747063,0.485356836663813,-0.509533392098773],[0,0,0,0],[8.999999E+09,8.999999E+09,8.999999E+09,8.999999E+09,8.999999E+09,8.999999E+09]];
    LOCAL CONST Robtarget Tr_meulage_bavure_48 := [[-104.3746328125,-49.837765625,96.85459375],[0.514201916085611,-0.490615999306146,0.48562952991373,-0.508975726724259],[0,0,0,0],[8.999999E+09,8.999999E+09,8.999999E+09,8.999999E+09,8.999999E+09,8.999999E+09]];
    LOCAL CONST Robtarget Tr_meulage_bavure_49 := [[-104.29021875,-57.2415078125,97.724328125],[0.513951818841022,-0.491197975096204,0.485900069155859,-0.508408497141546],[0,0,0,0],[8.999999E+09,8.999999E+09,8.999999E+09,8.999999E+09,8.999999E+09,8.999999E+09]];
    LOCAL CONST Robtarget Tr_meulage_bavure_50 := [[-104.2449609375,-60.18394921875,98.0699921875],[0.513701943556093,-0.491795928871391,0.486169582889697,-0.507824983833088],[0,0,0,0],[8.999999E+09,8.999999E+09,8.999999E+09,8.999999E+09,8.999999E+09,8.999999E+09]];
    LOCAL CONST Robtarget Tr_meulage_bavure_51 := [[-104.173984375,-62.51034765625,98.34328125],[0.513457319962121,-0.492416131349672,0.48643311678359,-0.507218648178615],[0,0,0,0],[8.999999E+09,8.999999E+09,8.999999E+09,8.999999E+09,8.999999E+09,8.999999E+09]];
    LOCAL CONST Robtarget Tr_meulage_bavure_52 := [[-104.21234375,-66.146703125,98.770453125],[0.513230412934505,-0.49305952983543,0.486678074550635,-0.506587894673005],[0,0,0,0],[8.999999E+09,8.999999E+09,8.999999E+09,8.999999E+09,8.999999E+09,8.999999E+09]];
    LOCAL CONST Robtarget Tr_meulage_bavure_53 := [[-104.21234375,-66.14671875,98.770453125],[0.513015983384075,-0.493734568640113,0.486909715366461,-0.505924604663565],[0,0,0,0],[8.999999E+09,8.999999E+09,8.999999E+09,8.999999E+09,8.999999E+09,8.999999E+09]];
    LOCAL CONST Robtarget Tr_meulage_bavure_54 := [[-104.1104453125,-72.6128203125,99.530046875],[0.512806343326415,-0.494439565482004,0.487135428719142,-0.505230882287272],[0,0,0,0],[8.999999E+09,8.999999E+09,8.999999E+09,8.999999E+09,8.999999E+09,8.999999E+09]];
    LOCAL CONST Robtarget Tr_meulage_bavure_55 := [[-104.0638125,-80.1904375,100.4202109375],[0.512599983496943,-0.495155888592037,0.487356121345882,-0.504525434342276],[0,0,0,0],[8.999999E+09,8.999999E+09,8.999999E+09,8.999999E+09,8.999999E+09,8.999999E+09]];
    LOCAL CONST Robtarget Tr_meulage_bavure_56 := [[-104.0132734375,-82.6676875,100.71121875],[0.512374902033798,-0.495874674565425,0.487593547507386,-0.503818220511776],[0,0,0,0],[8.999999E+09,8.999999E+09,8.999999E+09,8.999999E+09,8.999999E+09,8.999999E+09]];
    LOCAL CONST Robtarget Tr_meulage_bavure_57 := [[-103.944,-84.3781171875,100.9121484375],[0.512116598536175,-0.496581585343533,0.487861998144621,-0.503124228563661],[0,0,0,0],[8.999999E+09,8.999999E+09,8.999999E+09,8.999999E+09,8.999999E+09,8.999999E+09]];
    LOCAL CONST Robtarget Tr_meulage_bavure_58 := [[-103.9050625,-85.7278125,101.070703125],[0.511812223183382,-0.497261248780204,0.488174266671599,-0.50245933568925],[0,0,0,0],[8.999999E+09,8.999999E+09,8.999999E+09,8.999999E+09,8.999999E+09,8.999999E+09]];
    LOCAL CONST Robtarget Tr_meulage_bavure_59 := [[-103.93875,-86.3869609375,101.1481328125],[0.511451504737901,-0.497912777240913,0.488540843509987,-0.501824739111304],[0,0,0,0],[8.999999E+09,8.999999E+09,8.999999E+09,8.999999E+09,8.999999E+09,8.999999E+09]];
    LOCAL CONST Robtarget Tr_meulage_bavure_60 := [[-103.7529921875,-95.482375,102.2166015625],[0.511038939871233,-0.498533504229751,0.488957444316439,-0.501222669821734],[0,0,0,0],[8.999999E+09,8.999999E+09,8.999999E+09,8.999999E+09,8.999999E+09,8.999999E+09]];
    LOCAL CONST Robtarget Tr_meulage_bavure_61 := [[-103.7406328125,-97.6751015625,102.4741875],[0.510578362561507,-0.499130982987864,0.489420491065473,-0.500645164193973],[0,0,0,0],[8.999999E+09,8.999999E+09,8.999999E+09,8.999999E+09,8.999999E+09,8.999999E+09]];
    LOCAL CONST Robtarget Tr_meulage_bavure_62 := [[-103.7224140625,-98.4227890625,102.5620234375],[0.51008205125636,-0.499722418171092,0.489917886845755,-0.50007426439673],[0,0,0,0],[8.999999E+09,8.999999E+09,8.999999E+09,8.999999E+09,8.999999E+09,8.999999E+09]];
    LOCAL CONST Robtarget Tr_meulage_bavure_63 := [[-103.6572578125,-105.02315625,103.3373828125],[0.509569681792752,-0.500317816049661,0.490429982979899,-0.499499003137411],[0,0,0,0],[8.999999E+09,8.999999E+09,8.999999E+09,8.999999E+09,8.999999E+09,8.999999E+09]];
    LOCAL CONST Robtarget Tr_meulage_bavure_64 := [[-103.6298828125,-106.490078125,103.5097109375],[0.509056882473052,-0.500932423304275,0.490941059202532,-0.498903471704117],[0,0,0,0],[8.999999E+09,8.999999E+09,8.999999E+09,8.999999E+09,8.999999E+09,8.999999E+09]];
    LOCAL CONST Robtarget Tr_meulage_bavure_65 := [[-103.6533828125,-106.90859375,103.558875],[0.508554227596862,-0.501581347808002,0.491440297152452,-0.498272198159978],[0,0,0,0],[8.999999E+09,8.999999E+09,8.999999E+09,8.999999E+09,8.999999E+09,8.999999E+09]];
    LOCAL CONST Robtarget Tr_meulage_bavure_66 := [[-103.6365078125,-107.7107578125,103.653109375],[0.508064424791715,-0.502272087201559,0.491924650005127,-0.497597658150223],[0,0,0,0],[8.999999E+09,8.999999E+09,8.999999E+09,8.999999E+09,8.999999E+09,8.999999E+09]];
    LOCAL CONST Robtarget Tr_meulage_bavure_67 := [[-103.62378125,-109.5723046875,103.8717890625],[0.50758825871173,-0.503003901748732,0.492392993967061,-0.496880643551043],[0,0,0,0],[8.999999E+09,8.999999E+09,8.999999E+09,8.999999E+09,8.999999E+09,8.999999E+09]];
    LOCAL CONST Robtarget Tr_meulage_bavure_68 := [[-103.54953125,-110.3712890625,103.9656484375],[0.507121355411283,-0.503764679888296,0.492849526500729,-0.496133472374997],[0,0,0,0],[8.999999E+09,8.999999E+09,8.999999E+09,8.999999E+09,8.999999E+09,8.999999E+09]];
    LOCAL CONST Robtarget Tr_meulage_bavure_69 := [[-103.5324375,-113.253640625,104.3042421875],[0.506659139114465,-0.504551663431849,0.493298608204174,-0.495359080691743],[0,0,0,0],[8.999999E+09,8.999999E+09,8.999999E+09,8.999999E+09,8.999999E+09,8.999999E+09]];
    LOCAL CONST Robtarget Tr_meulage_bavure_70 := [[-103.42459375,-117.5753984375,104.8119375],[0.506174661297521,-0.505349584852028,0.493767274373848,-0.494573440560292],[0,0,0,0],[8.999999E+09,8.999999E+09,8.999999E+09,8.999999E+09,8.999999E+09,8.999999E+09]];
    LOCAL CONST Robtarget Tr_meulage_bavure_71 := [[-103.3727109375,-119.2358671875,105.0069921875],[0.505649774039922,-0.506125182043875,0.494274392661514,-0.493810116212215],[0,0,0,0],[8.999999E+09,8.999999E+09,8.999999E+09,8.999999E+09,8.999999E+09,8.999999E+09]];
    LOCAL CONST Robtarget Tr_meulage_bavure_72 := [[-103.380890625,-120.229109375,105.123671875],[0.505080893825889,-0.506882874732621,0.494823628126536,-0.493064518133811],[0,0,0,0],[8.999999E+09,8.999999E+09,8.999999E+09,8.999999E+09,8.999999E+09,8.999999E+09]];
    LOCAL CONST Robtarget Tr_meulage_bavure_73 := [[-103.241609375,-128.01434375,106.0382265625],[0.504468733555157,-0.507621251309311,0.495414467039611,-0.492337757979502],[0,0,0,0],[8.999999E+09,8.999999E+09,8.999999E+09,8.999999E+09,8.999999E+09,8.999999E+09]];
    LOCAL CONST Robtarget Tr_meulage_bavure_74 := [[-103.1030859375,-133.25215625,106.65353125],[0.50383993236617,-0.508368173831336,0.496019492819809,-0.491601246063744],[0,0,0,0],[8.999999E+09,8.999999E+09,8.999999E+09,8.999999E+09,8.999999E+09,8.999999E+09]];
    LOCAL CONST Robtarget Tr_meulage_bavure_75 := [[-103.0835546875,-135.7205,106.9434921875],[0.50324297509514,-0.509164421235232,0.496588631440712,-0.490813438374934],[0,0,0,0],[8.999999E+09,8.999999E+09,8.999999E+09,8.999999E+09,8.999999E+09,8.999999E+09]];
    LOCAL CONST Robtarget Tr_meulage_bavure_76 := [[-103.0544453125,-136.87503125,107.079125],[0.50276977529987,-0.510100907369252,0.497025813749839,-0.489882595947534],[0,0,0,0],[8.999999E+09,8.999999E+09,8.999999E+09,8.999999E+09,8.999999E+09,8.999999E+09]];
    LOCAL CONST Robtarget Tr_meulage_bavure_77 := [[-103.03140625,-137.77490625,107.1848359375],[0.502547973113544,-0.511310033343984,0.49719583627619,-0.488675643869082],[0,0,0,0],[8.999999E+09,8.999999E+09,8.999999E+09,8.999999E+09,8.999999E+09,8.999999E+09]];
    LOCAL CONST Robtarget Tr_meulage_bavure_78 := [[-103.0259375,-138.63625,107.286015625],[0.502732314930253,-0.512959225427248,0.496931309203267,-0.487023948597473],[0,0,0,0],[8.999999E+09,8.999999E+09,8.999999E+09,8.999999E+09,8.999999E+09,8.999999E+09]];
    LOCAL CONST Robtarget Tr_meulage_bavure_79 := [[-102.9553828125,-147.00771875,108.2694375],[0.503559973557534,-0.515281514335282,0.495971987252347,-0.484689696482225],[0,0,0,0],[8.999999E+09,8.999999E+09,8.999999E+09,8.999999E+09,8.999999E+09,8.999999E+09]];
    LOCAL CONST Robtarget Tr_meulage_bavure_80 := [[-102.9019453125,-152.602734375,108.926703125],[0.50526978977669,-0.518539560969587,0.494040201557502,-0.481397385216735],[0,0,0,0],[8.999999E+09,8.999999E+09,8.999999E+09,8.999999E+09,8.999999E+09,8.999999E+09]];
    LOCAL CONST Robtarget Tr_meulage_bavure_81 := [[-102.8525703125,-157.765171875,109.5331484375],[0.508142259942592,-0.523016913966868,0.490790672352161,-0.476832535904507],[0,0,0,0],[8.999999E+09,8.999999E+09,8.999999E+09,8.999999E+09,8.999999E+09,8.999999E+09]];
    LOCAL CONST Robtarget Tr_meulage_bavure_82 := [[-102.85928125,-158.70746875,109.64384375],[0.512449290499543,-0.529004866091056,0.485846098262,-0.470641206357975],[0,0,0,0],[8.999999E+09,8.999999E+09,8.999999E+09,8.999999E+09,8.999999E+09,8.999999E+09]];
    LOCAL CONST Robtarget Tr_meulage_bavure_83 := [[-102.677796875,-171.792984375,111.1810390625],[0.518414199966014,-0.536741707812304,0.478824162733193,-0.462474299341257],[0,0,0,0],[8.999999E+09,8.999999E+09,8.999999E+09,8.999999E+09,8.999999E+09,8.999999E+09]];
    LOCAL CONST Robtarget Tr_meulage_bavure_84 := [[-102.6637578125,-177.023328125,111.7954609375],[0.526173057629139,-0.546392116880473,0.469361355569094,-0.451992794117806],[0,0,0,0],[8.999999E+09,8.999999E+09,8.999999E+09,8.999999E+09,8.999999E+09,8.999999E+09]];
    LOCAL CONST Robtarget Tr_meulage_bavure_85 := [[-102.6677890625,-177.957,111.905140625],[0.535769187405778,-0.558012100198399,0.457110364615404,-0.438889494542643],[0,0,0,0],[8.999999E+09,8.999999E+09,8.999999E+09,8.999999E+09,8.999999E+09,8.999999E+09]];
    LOCAL CONST Robtarget Tr_meulage_bavure_86 := [[-102.7553125,-179.215171875,112.0529453125],[0.547118265385656,-0.571531669198047,0.441774999894637,-0.422904249509482],[0,0,0,0],[8.999999E+09,8.999999E+09,8.999999E+09,8.999999E+09,8.999999E+09,8.999999E+09]];
    LOCAL CONST Robtarget Tr_meulage_bavure_87 := [[-102.7847578125,-180.26753125,112.1765703125],[0.559991391437042,-0.586705488029073,0.423155523263219,-0.403888245638325],[0,0,0,0],[8.999999E+09,8.999999E+09,8.999999E+09,8.999999E+09,8.999999E+09,8.999999E+09]];
    LOCAL CONST Robtarget Tr_meulage_bavure_88 := [[-102.1311015625,-184.77121875,112.7056328125],[0.574021923674172,-0.603175640692349,0.401159971635054,-0.381770421555339],[0,0,0,0],[8.999999E+09,8.999999E+09,8.999999E+09,8.999999E+09,8.999999E+09,8.999999E+09]];
    LOCAL CONST Robtarget Tr_meulage_bavure_89 := [[-102.10940625,-184.901390625,112.720921875],[0.588753204392245,-0.620461563236625,0.375808066108009,-0.356602594370801],[0,0,0,0],[8.999999E+09,8.999999E+09,8.999999E+09,8.999999E+09,8.999999E+09,8.999999E+09]];
    LOCAL CONST Robtarget Tr_meulage_bavure_90 := [[-101.9547421875,-185.108140625,112.7452109375],[0.60365108993816,-0.638010758937903,0.347265635240582,-0.328563862402589],[0,0,0,0],[8.999999E+09,8.999999E+09,8.999999E+09,8.999999E+09,8.999999E+09,8.999999E+09]];
    LOCAL CONST Robtarget Tr_meulage_bavure_91 := [[-100.387484375,-187.2984375,113.0025078125],[0.6181419491209,-0.655203923722824,0.315894219637126,-0.298025487291074],[0,0,0,0],[8.999999E+09,8.999999E+09,8.999999E+09,8.999999E+09,8.999999E+09,8.999999E+09]];
    LOCAL CONST Robtarget Tr_meulage_bavure_92 := [[-99.3960859375,-187.773046875,113.058265625],[0.631657020525799,-0.671437193591113,0.282260774641173,-0.265537866568831],[0,0,0,0],[8.999999E+09,8.999999E+09,8.999999E+09,8.999999E+09,8.999999E+09,8.999999E+09]];
    LOCAL CONST Robtarget Tr_meulage_bavure_93 := [[-96.7586328125,-188.415203125,113.133703125],[0.64368713356643,-0.686148026820319,0.247179707284045,-0.231883487291761],[0,0,0,0],[8.999999E+09,8.999999E+09,8.999999E+09,8.999999E+09,8.999999E+09,8.999999E+09]];
    LOCAL CONST Robtarget Tr_meulage_bavure_94 := [[-96.5877109375,-188.470890625,113.1402421875],[0.653828991432091,-0.698877825246834,0.211744242123502,-0.198095459990114],[0,0,0,0],[8.999999E+09,8.999999E+09,8.999999E+09,8.999999E+09,8.999999E+09,8.999999E+09]];
    LOCAL CONST Robtarget Tr_meulage_bavure_95 := [[-95.7683125,-188.576609375,113.1526640625],[0.661866365126718,-0.709378211754516,0.177171411528397,-0.16530504632027],[0,0,0,0],[8.999999E+09,8.999999E+09,8.999999E+09,8.999999E+09,8.999999E+09,8.999999E+09]];
    LOCAL CONST Robtarget Tr_meulage_bavure_96 := [[-92.7172265625,-188.44696875,113.1374296875],[0.667799725354698,-0.717639099090743,0.144642107356311,-0.134596846367],[0,0,0,0],[8.999999E+09,8.999999E+09,8.999999E+09,8.999999E+09,8.999999E+09,8.999999E+09]];
    LOCAL CONST Robtarget Tr_meulage_bavure_97 := [[-89.9671015625,-188.451375,113.1379453125],[0.671838850623296,-0.723852080018129,0.115123809796233,-0.106851455135611],[0,0,0,0],[8.999999E+09,8.999999E+09,8.999999E+09,8.999999E+09,8.999999E+09,8.999999E+09]];
    LOCAL CONST Robtarget Tr_meulage_bavure_98 := [[-86.339234375,-188.310671875,113.121421875],[0.674319366758754,-0.728357875178739,0.0892354945883128,-0.0826149126051926],[0,0,0,0],[8.999999E+09,8.999999E+09,8.999999E+09,8.999999E+09,8.999999E+09,8.999999E+09]];
    LOCAL CONST Robtarget Tr_meulage_bavure_99 := [[-83.283265625,-188.283078125,113.1181796875],[0.675619859255385,-0.731551759957692,0.0672091599718059,-0.0620705815859841],[0,0,0,0],[8.999999E+09,8.999999E+09,8.999999E+09,8.999999E+09,8.999999E+09,8.999999E+09]];
    LOCAL CONST Robtarget Tr_meulage_bavure_100 := [[-79.7990078125,-188.25809375,113.1152421875],[0.676093729750279,-0.733800985164171,0.0489678168253839,-0.0451169112396263],[0,0,0,0],[8.999999E+09,8.999999E+09,8.999999E+09,8.999999E+09,8.999999E+09,8.999999E+09]];
    LOCAL CONST Robtarget Tr_meulage_bavure_101 := [[-78.6981171875,-188.25709375,113.115125],[0.676026898389928,-0.735409421220669,0.0342206020383296,-0.0314573716211155],[0,0,0,0],[8.999999E+09,8.999999E+09,8.999999E+09,8.999999E+09,8.999999E+09,8.999999E+09]];
    LOCAL CONST Robtarget Tr_meulage_bavure_102 := [[-78.0926484375,-188.29284375,113.119328125],[0.67563535223383,-0.736599721911609,0.0225669035520712,-0.0206991631637625],[0,0,0,0],[8.999999E+09,8.999999E+09,8.999999E+09,8.999999E+09,8.999999E+09,8.999999E+09]];
    LOCAL CONST Robtarget Tr_meulage_bavure_103 := [[-76.498140625,-188.382390625,113.12984375],[0.675061121345871,-0.737533037668524,0.0135516500718072,-0.0124037726126549],[0,0,0,0],[8.999999E+09,8.999999E+09,8.999999E+09,8.999999E+09,8.999999E+09,8.999999E+09]];
    LOCAL CONST Robtarget Tr_meulage_bavure_104 := [[-71.1280859375,-188.79228125,113.1779921875],[0.674402293347765,-0.738307725913775,0.0067366489522568,-0.00615354728579854],[0,0,0,0],[8.999999E+09,8.999999E+09,8.999999E+09,8.999999E+09,8.999999E+09,8.999999E+09]];
    LOCAL CONST Robtarget Tr_meulage_bavure_105 := [[-70.5999765625,-188.812984375,113.1804296875],[0.67372470626486,-0.738978635480716,0.00174819648167075,-0.00159382572723596],[0,0,0,0],[8.999999E+09,8.999999E+09,8.999999E+09,8.999999E+09,8.999999E+09,8.999999E+09]];
    LOCAL CONST Robtarget Tr_meulage_bavure_106 := [[-69.4306640625,-188.84671875,113.184390625],[0.673056374859989,-0.739587349497377,-0.00176089456347665,0.00160248997256336],[0,0,0,0],[8.999999E+09,8.999999E+09,8.999999E+09,8.999999E+09,8.999999E+09,8.999999E+09]];
    LOCAL CONST Robtarget Tr_meulage_bavure_107 := [[-62.37869140625,-188.349828125,113.1260234375],[0.672420039749452,-0.740149353293788,-0.00406919788498653,0.0036968352284501],[0,0,0,0],[8.999999E+09,8.999999E+09,8.999999E+09,8.999999E+09,8.999999E+09,8.999999E+09]];
    LOCAL CONST Robtarget Tr_meulage_bavure_108 := [[-60.9710390625,-188.2785625,113.1176484375],[0.671825709534592,-0.740673077815688,-0.00542315756183196,0.00491906184526162],[0,0,0,0],[8.999999E+09,8.999999E+09,8.999999E+09,8.999999E+09,8.999999E+09,8.999999E+09]];
    LOCAL CONST Robtarget Tr_meulage_bavure_109 := [[-55.11535546875,-188.014578125,113.0866328125],[0.671273759793528,-0.741164382326639,-0.0060622651917143,0.00549060322533692],[0,0,0,0],[8.999999E+09,8.999999E+09,8.999999E+09,8.999999E+09,8.999999E+09,8.999999E+09]];
    LOCAL CONST Robtarget Tr_meulage_bavure_110 := [[-54.10494921875,-187.99359375,113.084171875],[0.67076755259017,-0.741620803716333,-0.00618169809007683,0.00559110866085975],[0,0,0,0],[8.999999E+09,8.999999E+09,8.999999E+09,8.999999E+09,8.999999E+09,8.999999E+09]];
    LOCAL CONST Robtarget Tr_meulage_bavure_111 := [[-51.1435859375,-188.006015625,113.0856328125],[0.670307732700726,-0.742039650574835,-0.00596890730202788,0.00539190152065818],[0,0,0,0],[8.999999E+09,8.999999E+09,8.999999E+09,8.999999E+09,8.999999E+09,8.999999E+09]];
    LOCAL CONST Robtarget Tr_meulage_bavure_112 := [[-50.70300390625,-188.02090625,113.0873828125],[0.669892418640747,-0.74242006649715,-0.00558522536526865,0.00503959994810812],[0,0,0,0],[8.999999E+09,8.999999E+09,8.999999E+09,8.999999E+09,8.999999E+09,8.999999E+09]];
    LOCAL CONST Robtarget Tr_meulage_bavure_113 := [[-49.09527734375,-188.076953125,113.0939609375],[0.669522112133806,-0.742759647494023,-0.0051593598397262,0.00465063699785821],[0,0,0,0],[8.999999E+09,8.999999E+09,8.999999E+09,8.999999E+09,8.999999E+09,8.999999E+09]];
    LOCAL CONST Robtarget Tr_meulage_bavure_114 := [[-41.8825078125,-188.36571875,113.127890625],[0.669195649658089,-0.743058509990707,-0.0047715066597723,0.00429720063238917],[0,0,0,0],[8.999999E+09,8.999999E+09,8.999999E+09,8.999999E+09,8.999999E+09,8.999999E+09]];
    LOCAL CONST Robtarget Tr_meulage_bavure_115 := [[-36.25433203125,-188.238015625,113.1128828125],[0.668915468035016,-0.743314302457776,-0.0044565196380904,0.00401046355446634],[0,0,0,0],[8.999999E+09,8.999999E+09,8.999999E+09,8.999999E+09,8.999999E+09,8.999999E+09]];
    LOCAL CONST Robtarget Tr_meulage_bavure_116 := [[-34.71267578125,-188.19140625,113.10740625],[0.668681309577192,-0.743527303926472,-0.00423586084378487,0.00380946464407031],[0,0,0,0],[8.999999E+09,8.999999E+09,8.999999E+09,8.999999E+09,8.999999E+09,8.999999E+09]];
    LOCAL CONST Robtarget Tr_meulage_bavure_117 := [[-29.997314453125,-188.079390625,113.09425],[0.668492852999227,-0.743698041011284,-0.00410924072024621,0.00369370080496999],[0,0,0,0],[8.999999E+09,8.999999E+09,8.999999E+09,8.999999E+09,8.999999E+09,8.999999E+09]];
    LOCAL CONST Robtarget Tr_meulage_bavure_118 := [[-29.189544921875,-188.102390625,113.096953125],[0.668352031483011,-0.743825068227274,-0.004062591061259,0.00365037574674419],[0,0,0,0],[8.999999E+09,8.999999E+09,8.999999E+09,8.999999E+09,8.999999E+09,8.999999E+09]];
    LOCAL CONST Robtarget Tr_meulage_bavure_119 := [[-23.36901953125,-188.123625,113.0994453125],[0.668256945494993,-0.743910371827088,-0.00407554178412953,0.00366107155786861],[0,0,0,0],[8.999999E+09,8.999999E+09,8.999999E+09,8.999999E+09,8.999999E+09,8.999999E+09]];
    LOCAL CONST Robtarget Tr_meulage_bavure_120 := [[-23.10696484375,-188.1266875,113.0998046875],[0.668209052604531,-0.743952872609388,-0.00412785262249192,0.00370758497173608],[0,0,0,0],[8.999999E+09,8.999999E+09,8.999999E+09,8.999999E+09,8.999999E+09,8.999999E+09]];
    LOCAL CONST Robtarget Tr_meulage_bavure_121 := [[-18.19451953125,-187.9670625,113.0810546875],[0.668208714675254,-0.743952424730657,-0.0042021385523808,0.0037743080170621],[0,0,0,0],[8.999999E+09,8.999999E+09,8.999999E+09,8.999999E+09,8.999999E+09,8.999999E+09]];
    LOCAL CONST Robtarget Tr_meulage_bavure_122 := [[-16.1770625,-187.919609375,113.0754765625],[0.668252985633157,-0.743911766570029,-0.00428843392004356,0.00385228315983337],[0,0,0,0],[8.999999E+09,8.999999E+09,8.999999E+09,8.999999E+09,8.999999E+09,8.999999E+09]];
    LOCAL CONST Robtarget Tr_meulage_bavure_123 := [[-10.464751953125,-187.93484375,113.0772734375],[0.668346232968856,-0.743827100845064,-0.00437267344794271,0.0039289504558455],[0,0,0,0],[8.999999E+09,8.999999E+09,8.999999E+09,8.999999E+09,8.999999E+09,8.999999E+09]];
    LOCAL CONST Robtarget Tr_meulage_bavure_124 := [[-9.772552734375,-187.9214375,113.0756953125],[0.668482650273322,-0.743703792327514,-0.00443841212893086,0.00398949357736547],[0,0,0,0],[8.999999E+09,8.999999E+09,8.999999E+09,8.999999E+09,8.999999E+09,8.999999E+09]];
    LOCAL CONST Robtarget Tr_meulage_bavure_125 := [[0.806488037109375,-187.835828125,113.065640625],[0.668664229066353,-0.743540096437968,-0.00447825206344311,0.00402728377112721],[0,0,0,0],[8.999999E+09,8.999999E+09,8.999999E+09,8.999999E+09,8.999999E+09,8.999999E+09]];
    LOCAL CONST Robtarget Tr_meulage_bavure_126 := [[2.207763671875,-187.8066875,113.06221875],[0.66888892092132,-0.743337899776254,-0.00448347681079243,0.00403443436268943],[0,0,0,0],[8.999999E+09,8.999999E+09,8.999999E+09,8.999999E+09,8.999999E+09,8.999999E+09]];
    LOCAL CONST Robtarget Tr_meulage_bavure_127 := [[6.42486572265625,-187.6513125,113.0439609375],[0.669157627514984,-0.743096353366077,-0.00445116824096168,0.00400827317520778],[0,0,0,0],[8.999999E+09,8.999999E+09,8.999999E+09,8.999999E+09,8.999999E+09,8.999999E+09]];
    LOCAL CONST Robtarget Tr_meulage_bavure_128 := [[10.275451171875,-187.683640625,113.0477578125],[0.66946709510536,-0.742818230665511,-0.00438740789364518,0.00395416414991515],[0,0,0,0],[8.999999E+09,8.999999E+09,8.999999E+09,8.999999E+09,8.999999E+09,8.999999E+09]];
    LOCAL CONST Robtarget Tr_meulage_bavure_129 := [[13.6043701171875,-187.719171875,113.0519375],[0.669819807973456,-0.742501004486747,-0.00430934157707945,0.00388751305413609],[0,0,0,0],[8.999999E+09,8.999999E+09,8.999999E+09,8.999999E+09,8.999999E+09,8.999999E+09]];
    LOCAL CONST Robtarget Tr_meulage_bavure_130 := [[16.82894921875,-187.69034375,113.048546875],[0.670211440362136,-0.742148206708157,-0.00424165811107748,0.0038305122433138],[0,0,0,0],[8.999999E+09,8.999999E+09,8.999999E+09,8.999999E+09,8.999999E+09,8.999999E+09]];
    LOCAL CONST Robtarget Tr_meulage_bavure_131 := [[19.891357421875,-187.64171875,113.0428359375],[0.670642278855219,-0.741759241996736,-0.00420661591362668,0.00380330209973391],[0,0,0,0],[8.999999E+09,8.999999E+09,8.999999E+09,8.999999E+09,8.999999E+09,8.999999E+09]];
    LOCAL CONST Robtarget Tr_meulage_bavure_132 := [[22.2802421875,-187.6446875,113.0431875],[0.67110766301019,-0.741338016319137,-0.00422310682691769,0.00382303253153961],[0,0,0,0],[8.999999E+09,8.999999E+09,8.999999E+09,8.999999E+09,8.999999E+09,8.999999E+09]];
    LOCAL CONST Robtarget Tr_meulage_bavure_133 := [[23.846771484375,-187.67796875,113.04709375],[0.671610800862882,-0.740881389177172,-0.00430097254453498,0.00389884218624047],[0,0,0,0],[8.999999E+09,8.999999E+09,8.999999E+09,8.999999E+09,8.999999E+09,8.999999E+09]];
    LOCAL CONST Robtarget Tr_meulage_bavure_134 := [[25.43017578125,-187.602921875,113.03828125],[0.672146452949343,-0.740393965004214,-0.00443765136190025,0.00402860066844291],[0,0,0,0],[8.999999E+09,8.999999E+09,8.999999E+09,8.999999E+09,8.999999E+09,8.999999E+09]];
    LOCAL CONST Robtarget Tr_meulage_bavure_135 := [[30.425048828125,-187.560609375,113.0333046875],[0.672714167854617,-0.73987582879663,-0.00464462218777852,0.00422301017068277],[0,0,0,0],[8.999999E+09,8.999999E+09,8.999999E+09,8.999999E+09,8.999999E+09,8.999999E+09]];
    LOCAL CONST Robtarget Tr_meulage_bavure_136 := [[35.5959453125,-187.47615625,113.0233828125],[0.673314202176167,-0.739326790139379,-0.00489769574400256,0.00446039308511058],[0,0,0,0],[8.999999E+09,8.999999E+09,8.999999E+09,8.999999E+09,8.999999E+09,8.999999E+09]];
    LOCAL CONST Robtarget Tr_meulage_bavure_137 := [[36.2562265625,-187.48925,113.024921875],[0.673943839641821,-0.738749525517151,-0.00516289958872537,0.00470999202344662],[0,0,0,0],[8.999999E+09,8.999999E+09,8.999999E+09,8.999999E+09,8.999999E+09,8.999999E+09]];
    LOCAL CONST Robtarget Tr_meulage_bavure_138 := [[36.97543359375,-187.464015625,113.0219609375],[0.674599365674952,-0.738147004743274,-0.00545920526220337,0.00498921811415141],[0,0,0,0],[8.999999E+09,8.999999E+09,8.999999E+09,8.999999E+09,8.999999E+09,8.999999E+09]];
    LOCAL CONST Robtarget Tr_meulage_bavure_139 := [[42.651671875,-187.350609375,113.008640625],[0.675280385330943,-0.737519111852603,-0.0058055768789843,0.0053156482712172],[0,0,0,0],[8.999999E+09,8.999999E+09,8.999999E+09,8.999999E+09,8.999999E+09,8.999999E+09]];
    LOCAL CONST Robtarget Tr_meulage_bavure_140 := [[45.55154296875,-187.41125,113.015765625],[0.675984267277483,-0.736866790573196,-0.00627889269744191,0.00576010852123291],[0,0,0,0],[8.999999E+09,8.999999E+09,8.999999E+09,8.999999E+09,8.999999E+09,8.999999E+09]];
    LOCAL CONST Robtarget Tr_meulage_bavure_141 := [[47.837921875,-187.44334375,113.01953125],[0.676708747361639,-0.736189684986152,-0.00698515877372108,0.00642078820212738],[0,0,0,0],[8.999999E+09,8.999999E+09,8.999999E+09,8.999999E+09,8.999999E+09,8.999999E+09]];
    LOCAL CONST Robtarget Tr_meulage_bavure_142 := [[48.56747265625,-187.432171875,113.01821875],[0.677447493528782,-0.735488334677671,-0.00811766916136998,0.00747706573629894],[0,0,0,0],[8.999999E+09,8.999999E+09,8.999999E+09,8.999999E+09,8.999999E+09,8.999999E+09]];
    LOCAL CONST Robtarget Tr_meulage_bavure_143 := [[50.01123046875,-187.409859375,113.0156015625],[0.678193682939999,-0.734757964066251,-0.00996935642598563,0.00920187991384754],[0,0,0,0],[8.999999E+09,8.999999E+09,8.999999E+09,8.999999E+09,8.999999E+09,8.999999E+09]];
    LOCAL CONST Robtarget Tr_meulage_bavure_144 := [[56.44015625,-187.30696875,113.003515625],[0.678934494105832,-0.73398848149993,-0.0129014457150598,0.0119337520145932],[0,0,0,0],[8.999999E+09,8.999999E+09,8.999999E+09,8.999999E+09,8.999999E+09,8.999999E+09]];
    LOCAL CONST Robtarget Tr_meulage_bavure_145 := [[58.77712890625,-187.2440625,112.996125],[0.679644319104375,-0.733156777974083,-0.0174278248703471,0.016155783487684],[0,0,0,0],[8.999999E+09,8.999999E+09,8.999999E+09,8.999999E+09,8.999999E+09,8.999999E+09]];
    LOCAL CONST Robtarget Tr_meulage_bavure_146 := [[60.86306640625,-187.234359375,112.994984375],[0.680276282398588,-0.732215699108842,-0.0241245536117678,0.0224132884142099],[0,0,0,0],[8.999999E+09,8.999999E+09,8.999999E+09,8.999999E+09,8.999999E+09,8.999999E+09]];
    LOCAL CONST Robtarget Tr_meulage_bavure_147 := [[68.35303125,-187.103328125,112.9795859375],[0.680743657678337,-0.731075107409365,-0.0336751332596861,0.0313567418117108],[0,0,0,0],[8.999999E+09,8.999999E+09,8.999999E+09,8.999999E+09,8.999999E+09,8.999999E+09]];
    LOCAL CONST Robtarget Tr_meulage_bavure_148 := [[68.5308203125,-187.104015625,112.979671875],[0.680890705871298,-0.72957534886487,-0.046855549991693,0.0437288740052274],[0,0,0,0],[8.999999E+09,8.999999E+09,8.999999E+09,8.999999E+09,8.999999E+09,8.999999E+09]];
    LOCAL CONST Robtarget Tr_meulage_bavure_149 := [[74.826140625,-187.067171875,112.97534375],[0.68046414431475,-0.727453360425966,-0.0644162401955566,0.0602553292749602],[0,0,0,0],[8.999999E+09,8.999999E+09,8.999999E+09,8.999999E+09,8.999999E+09,8.999999E+09]];
    LOCAL CONST Robtarget Tr_meulage_bavure_150 := [[75.47121875,-187.060046875,112.9745078125],[0.679080303488451,-0.724304978700351,-0.0870303605997185,0.081596296348553],[0,0,0,0],[8.999999E+09,8.999999E+09,8.999999E+09,8.999999E+09,8.999999E+09,8.999999E+09]];
    LOCAL CONST Robtarget Tr_meulage_bavure_151 := [[77.0140390625,-187.093796875,112.97846875],[0.676197751578646,-0.719566130668737,-0.115178316701397,0.108236499002136],[0,0,0,0],[8.999999E+09,8.999999E+09,8.999999E+09,8.999999E+09,8.999999E+09,8.999999E+09]];
    LOCAL CONST Robtarget Tr_meulage_bavure_152 := [[80.16934375,-187.154828125,112.985640625],[0.671147691589279,-0.712540357516382,-0.148910143153902,0.140259702875388],[0,0,0,0],[8.999999E+09,8.999999E+09,8.999999E+09,8.999999E+09,8.999999E+09,8.999999E+09]];
    LOCAL CONST Robtarget Tr_meulage_bavure_153 := [[80.97790625,-187.181984375,112.988828125],[0.663247278031878,-0.702524553080736,-0.187600071913781,0.177111584940007],[0,0,0,0],[8.999999E+09,8.999999E+09,8.999999E+09,8.999999E+09,8.999999E+09,8.999999E+09]];
    LOCAL CONST Robtarget Tr_meulage_bavure_154 := [[82.5570390625,-186.745625,112.9375703125],[0.652021760304226,-0.689041408434497,-0.229794733203611,0.217448711525879],[0,0,0,0],[8.999999E+09,8.999999E+09,8.999999E+09,8.999999E+09,8.999999E+09,8.999999E+09]];
    LOCAL CONST Robtarget Tr_meulage_bavure_155 := [[84.562625,-185.99403125,112.8492734375],[0.637481858647314,-0.672130791493076,-0.273274737659092,0.259187184829442],[0,0,0,0],[8.999999E+09,8.999999E+09,8.999999E+09,8.999999E+09,8.999999E+09,8.999999E+09]];
    LOCAL CONST Robtarget Tr_meulage_bavure_156 := [[85.2157265625,-185.479359375,112.7888125],[0.620250120424451,-0.652471824825813,-0.315565302885759,0.299981408651513],[0,0,0,0],[8.999999E+09,8.999999E+09,8.999999E+09,8.999999E+09,8.999999E+09,8.999999E+09]];
    LOCAL CONST Robtarget Tr_meulage_bavure_157 := [[85.356875,-185.240984375,112.7608125],[0.601461183082971,-0.631276718506785,-0.354488363015397,0.337745688947175],[0,0,0,0],[8.999999E+09,8.999999E+09,8.999999E+09,8.999999E+09,8.999999E+09,8.999999E+09]];
    LOCAL CONST Robtarget Tr_meulage_bavure_158 := [[86.8857734375,-182.84078125,112.4788515625],[0.582431342266505,-0.609933905867462,-0.388630825437695,0.371107051318775],[0,0,0,0],[8.999999E+09,8.999999E+09,8.999999E+09,8.999999E+09,8.999999E+09,8.999999E+09]];
    LOCAL CONST Robtarget Tr_meulage_bavure_159 := [[87.516296875,-180.133796875,112.160859375],[0.56431692543511,-0.589655190194392,-0.41743695080885,0.399499131968631],[0,0,0,0],[8.999999E+09,8.999999E+09,8.999999E+09,8.999999E+09,8.999999E+09,8.999999E+09]];
    LOCAL CONST Robtarget Tr_meulage_bavure_160 := [[87.6045234375,-179.749125,112.115671875],[0.547967987943535,-0.571319245994112,-0.440962421481344,0.422939175517169],[0,0,0,0],[8.999999E+09,8.999999E+09,8.999999E+09,8.999999E+09,8.999999E+09,8.999999E+09]];
    LOCAL CONST Robtarget Tr_meulage_bavure_161 := [[87.62125,-179.313859375,112.0645390625],[0.533857456502739,-0.555407806621352,-0.459672412548169,0.441836686596564],[0,0,0,0],[8.999999E+09,8.999999E+09,8.999999E+09,8.999999E+09,8.999999E+09,8.999999E+09]];
    LOCAL CONST Robtarget Tr_meulage_bavure_162 := [[87.5428125,-176.117546875,111.6890546875],[0.522151420389827,-0.542079868360667,-0.474203043279391,0.456769946742922],[0,0,0,0],[8.999999E+09,8.999999E+09,8.999999E+09,8.999999E+09,8.999999E+09,8.999999E+09]];
    LOCAL CONST Robtarget Tr_meulage_bavure_163 := [[87.46734375,-174.9143125,111.5477109375],[0.512814827386339,-0.53127860845469,-0.485202579398711,0.468340100734504],[0,0,0,0],[8.999999E+09,8.999999E+09,8.999999E+09,8.999999E+09,8.999999E+09,8.999999E+09]];
    LOCAL CONST Robtarget Tr_meulage_bavure_164 := [[87.41675,-173.2148125,111.3480625],[0.505669341311933,-0.522805766275676,-0.493286407464658,0.477117562259734],[0,0,0,0],[8.999999E+09,8.999999E+09,8.999999E+09,8.999999E+09,8.999999E+09,8.999999E+09]];
    LOCAL CONST Robtarget Tr_meulage_bavure_165 := [[87.224703125,-165.819609375,110.479328125],[0.500455113965528,-0.516380530157976,-0.499008064108438,0.483618422864831],[0,0,0,0],[8.999999E+09,8.999999E+09,8.999999E+09,8.999999E+09,8.999999E+09,8.999999E+09]];
    LOCAL CONST Robtarget Tr_meulage_bavure_166 := [[87.1819140625,-154.80871875,109.18584375],[0.496879825831023,-0.511688062210159,-0.502846498852406,0.488294137037935],[0,0,0,0],[8.999999E+09,8.999999E+09,8.999999E+09,8.999999E+09,8.999999E+09,8.999999E+09]];
    LOCAL CONST Robtarget Tr_meulage_bavure_167 := [[87.13815625,-152.352046875,108.89725],[0.494615751404705,-0.508380941672057,-0.505242810108741,0.491562589545232],[0,0,0,0],[8.999999E+09,8.999999E+09,8.999999E+09,8.999999E+09,8.999999E+09,8.999999E+09]];
    LOCAL CONST Robtarget Tr_meulage_bavure_168 := [[87.1338828125,-151.900234375,108.8441796875],[0.4933642074842,-0.506148433956601,-0.506559108783672,0.493764509543831],[0,0,0,0],[8.999999E+09,8.999999E+09,8.999999E+09,8.999999E+09,8.999999E+09,8.999999E+09]];
    LOCAL CONST Robtarget Tr_meulage_bavure_169 := [[87.0577421875,-149.622734375,108.5766328125],[0.492873385652364,-0.504720528981122,-0.507081088501221,0.49517853651487],[0,0,0,0],[8.999999E+09,8.999999E+09,8.999999E+09,8.999999E+09,8.999999E+09,8.999999E+09]];
    LOCAL CONST Robtarget Tr_meulage_bavure_170 := [[86.9020703125,-143.449578125,107.851453125],[0.492903172933089,-0.503853191712713,-0.507066354427043,0.496046505401938],[0,0,0,0],[8.999999E+09,8.999999E+09,8.999999E+09,8.999999E+09,8.999999E+09,8.999999E+09]];
    LOCAL CONST Robtarget Tr_meulage_bavure_171 := [[86.8385625,-140.274109375,107.478421875],[0.493288135140607,-0.503370363178935,-0.506688536614456,0.496539847410166],[0,0,0,0],[8.999999E+09,8.999999E+09,8.999999E+09,8.999999E+09,8.999999E+09,8.999999E+09]];
    LOCAL CONST Robtarget Tr_meulage_bavure_172 := [[86.776125,-134.90296875,106.8474609375],[0.49388354535927,-0.503126903362148,-0.5060964302006,0.496798516578686],[0,0,0,0],[8.999999E+09,8.999999E+09,8.999999E+09,8.999999E+09,8.999999E+09,8.999999E+09]];
    LOCAL CONST Robtarget Tr_meulage_bavure_173 := [[86.7926015625,-131.294921875,106.423609375],[0.494601982303503,-0.503028175234433,-0.505379324408686,0.496913747527658],[0,0,0,0],[8.999999E+09,8.999999E+09,8.999999E+09,8.999999E+09,8.999999E+09,8.999999E+09]];
    LOCAL CONST Robtarget Tr_meulage_bavure_174 := [[86.6298203125,-125.8183515625,105.7802578125],[0.49538610799145,-0.503019274562131,-0.504595402827248,0.496938318983028],[0,0,0,0],[8.999999E+09,8.999999E+09,8.999999E+09,8.999999E+09,8.999999E+09,8.999999E+09]];
    LOCAL CONST Robtarget Tr_meulage_bavure_175 := [[86.57696875,-122.3426328125,105.371953125],[0.496181463697028,-0.503040165025452,-0.503799874046699,0.496930814465325],[0,0,0,0],[8.999999E+09,8.999999E+09,8.999999E+09,8.999999E+09,8.999999E+09,8.999999E+09]];
    LOCAL CONST Robtarget Tr_meulage_bavure_176 := [[86.74103125,-114.5384765625,104.4551796875],[0.49696174635949,-0.503067699841669,-0.503019319160516,0.4969139528959],[0,0,0,0],[8.999999E+09,8.999999E+09,8.999999E+09,8.999999E+09,8.999999E+09,8.999999E+09]];
    LOCAL CONST Robtarget Tr_meulage_bavure_177 := [[86.7685234375,-111.5094296875,104.09934375],[0.497704644606745,-0.5030728496944,-0.502276406122644,0.496916699749313],[0,0,0,0],[8.999999E+09,8.999999E+09,8.999999E+09,8.999999E+09,8.999999E+09,8.999999E+09]];
    LOCAL CONST Robtarget Tr_meulage_bavure_178 := [[86.636015625,-100.8385234375,102.8458046875],[0.498404123761893,-0.503053357141735,-0.501577199328827,0.496941608641316],[0,0,0,0],[8.999999E+09,8.999999E+09,8.999999E+09,8.999999E+09,8.999999E+09,8.999999E+09]];
    LOCAL CONST Robtarget Tr_meulage_bavure_179 := [[86.6317109375,-99.323671875,102.6678515625],[0.499062366905729,-0.503003688282826,-0.500919578282762,0.496994587098637],[0,0,0,0],[8.999999E+09,8.999999E+09,8.999999E+09,8.999999E+09,8.999999E+09,8.999999E+09]];
    LOCAL CONST Robtarget Tr_meulage_bavure_180 := [[86.6148359375,-90.64021875,101.64778125],[0.49966039086844,-0.502911644344964,-0.500322652365168,0.497088136359867],[0,0,0,0],[8.999999E+09,8.999999E+09,8.999999E+09,8.999999E+09,8.999999E+09,8.999999E+09]];
    LOCAL CONST Robtarget Tr_meulage_bavure_181 := [[86.621828125,-90.2091015625,101.5971328125],[0.500193840761526,-0.502771280883005,-0.499790798674857,0.49722863789553],[0,0,0,0],[8.999999E+09,8.999999E+09,8.999999E+09,8.999999E+09,8.999999E+09,8.999999E+09]];
    LOCAL CONST Robtarget Tr_meulage_bavure_182 := [[86.65240625,-88.2894140625,101.371625],[0.50066136614533,-0.502576785458611,-0.499325349520025,0.497422322070779],[0,0,0,0],[8.999999E+09,8.999999E+09,8.999999E+09,8.999999E+09,8.999999E+09,8.999999E+09]];
    LOCAL CONST Robtarget Tr_meulage_bavure_183 := [[86.72021875,-83.8615,100.8514609375],[0.501062294986018,-0.50232608334931,-0.498926873018206,0.497671636634601],[0,0,0,0],[8.999999E+09,8.999999E+09,8.999999E+09,8.999999E+09,8.999999E+09,8.999999E+09]];
    LOCAL CONST Robtarget Tr_meulage_bavure_184 := [[86.75509375,-82.858375,100.733625],[0.501395155621406,-0.502016056484893,-0.498596699581771,0.497980027829338],[0,0,0,0],[8.999999E+09,8.999999E+09,8.999999E+09,8.999999E+09,8.999999E+09,8.999999E+09]];
    LOCAL CONST Robtarget Tr_meulage_bavure_185 := [[86.7529296875,-82.0318046875,100.6365234375],[0.501657525865225,-0.501646153564295,-0.498337036311715,0.498348333595072],[0,0,0,0],[8.999999E+09,8.999999E+09,8.999999E+09,8.999999E+09,8.999999E+09,8.999999E+09]];
    LOCAL CONST Robtarget Tr_meulage_bavure_186 := [[86.7530546875,-81.27221875,100.5472890625],[0.501851883498429,-0.501213397483539,-0.498145155134743,0.498779732575282],[0,0,0,0],[8.999999E+09,8.999999E+09,8.999999E+09,8.999999E+09,8.999999E+09,8.999999E+09]];
    LOCAL CONST Robtarget Tr_meulage_bavure_187 := [[86.8179921875,-74.5208203125,99.7541875],[0.501975746338926,-0.500716901074738,-0.498023214535888,0.499275287640927],[0,0,0,0],[8.999999E+09,8.999999E+09,8.999999E+09,8.999999E+09,8.999999E+09,8.999999E+09]];
    LOCAL CONST Robtarget Tr_meulage_bavure_188 := [[86.8865078125,-71.090671875,99.351234375],[0.502030018484776,-0.500153649593467,-0.497969931732044,0.499838108220347],[0,0,0,0],[8.999999E+09,8.999999E+09,8.999999E+09,8.999999E+09,8.999999E+09,8.999999E+09]];
    LOCAL CONST Robtarget Tr_meulage_bavure_189 := [[86.900328125,-70.887234375,99.3273359375],[0.502011026886884,-0.499523294353891,-0.497988526297116,0.500468615357885],[0,0,0,0],[8.999999E+09,8.999999E+09,8.999999E+09,8.999999E+09,8.999999E+09,8.999999E+09]];
    LOCAL CONST Robtarget Tr_meulage_bavure_190 := [[86.8401171875,-65.770140625,98.72621875],[0.501920508047912,-0.498820741813358,-0.498076728044426,0.501171870836998],[0,0,0,0],[8.999999E+09,8.999999E+09,8.999999E+09,8.999999E+09,8.999999E+09,8.999999E+09]];
    LOCAL CONST Robtarget Tr_meulage_bavure_191 := [[86.8602265625,-65.12475390625,98.6503984375],[0.501755309706224,-0.498045320085184,-0.498237072893557,0.501948490900529],[0,0,0,0],[8.999999E+09,8.999999E+09,8.999999E+09,8.999999E+09,8.999999E+09,8.999999E+09]];
    LOCAL CONST Robtarget Tr_meulage_bavure_192 := [[86.8485078125,-64.69334765625,98.59971875],[0.501518058194156,-0.497195507450805,-0.498466237434781,0.502799835733379],[0,0,0,0],[8.999999E+09,8.999999E+09,8.999999E+09,8.999999E+09,8.999999E+09,8.999999E+09]];
    LOCAL CONST Robtarget Tr_meulage_bavure_193 := [[86.85146875,-64.3181953125,98.5556484375],[0.501212111858329,-0.496278302240927,-0.498760208059896,0.503718691838437],[0,0,0,0],[8.999999E+09,8.999999E+09,8.999999E+09,8.999999E+09,8.999999E+09,8.999999E+09]];
    LOCAL CONST Robtarget Tr_meulage_bavure_194 := [[86.83078125,-62.9726640625,98.3975859375],[0.500851938009311,-0.495299672685869,-0.499103889222866,0.504698799475684],[0,0,0,0],[8.999999E+09,8.999999E+09,8.999999E+09,8.999999E+09,8.999999E+09,8.999999E+09]];
    LOCAL CONST Robtarget Tr_meulage_bavure_195 := [[86.8465234375,-58.52182421875,97.874734375],[0.500457950199614,-0.494283627006954,-0.499476699328567,0.505715891566294],[0,0,0,0],[8.999999E+09,8.999999E+09,8.999999E+09,8.999999E+09,8.999999E+09,8.999999E+09]];
    LOCAL CONST Robtarget Tr_meulage_bavure_196 := [[86.850890625,-50.77744140625,96.9649765625],[0.500067142012504,-0.49326161501372,-0.499842042540759,0.506738359651394],[0,0,0,0],[8.999999E+09,8.999999E+09,8.999999E+09,8.999999E+09,8.999999E+09,8.999999E+09]];
    LOCAL CONST Robtarget Tr_meulage_bavure_197 := [[86.87615625,-48.06726953125,96.646609375],[0.499723790815913,-0.492277217648474,-0.50015692078353,0.507722688550737],[0,0,0,0],[8.999999E+09,8.999999E+09,8.999999E+09,8.999999E+09,8.999999E+09,8.999999E+09]];
    LOCAL CONST Robtarget Tr_meulage_bavure_198 := [[86.8739921875,-47.19005078125,96.5435546875],[0.49948137352002,-0.491382613285348,-0.500370103549159,0.508616991794041],[0,0,0,0],[8.999999E+09,8.999999E+09,8.999999E+09,8.999999E+09,8.999999E+09,8.999999E+09]];
    LOCAL CONST Robtarget Tr_meulage_bavure_199 := [[86.845578125,-46.0945234375,96.414859375],[0.49939776323434,-0.490635986186507,-0.500426861794835,0.509363484291429],[0,0,0,0],[8.999999E+09,8.999999E+09,8.999999E+09,8.999999E+09,8.999999E+09,8.999999E+09]];
    LOCAL CONST Robtarget Tr_meulage_bavure_200 := [[86.757140625,-40.4277578125,95.749171875],[0.499524976484677,-0.49008132157162,-0.500278249419788,0.509918394718282],[0,0,0,0],[8.999999E+09,8.999999E+09,8.999999E+09,8.999999E+09,8.999999E+09,8.999999E+09]];
    LOCAL CONST Robtarget Tr_meulage_bavure_201 := [[86.5478203125,-37.73457421875,95.432796875],[0.499895683495639,-0.489751897256471,-0.499894247220147,0.510248102742497],[0,0,0,0],[8.999999E+09,8.999999E+09,8.999999E+09,8.999999E+09,8.999999E+09,8.999999E+09]];
    LOCAL CONST Robtarget Tr_meulage_bavure_202 := [[86.445984375,-34.77364453125,95.0849609375],[0.500523044646909,-0.489654381772661,-0.499262885235623,0.510344824226153],[0,0,0,0],[8.999999E+09,8.999999E+09,8.999999E+09,8.999999E+09,8.999999E+09,8.999999E+09]];
    LOCAL CONST Robtarget Tr_meulage_bavure_203 := [[86.3346875,-33.1018828125,94.888578125],[0.501376720577843,-0.489766503783455,-0.498413898435749,0.51022910704939],[0,0,0,0],[8.999999E+09,8.999999E+09,8.999999E+09,8.999999E+09,8.999999E+09,8.999999E+09]];
    LOCAL CONST Robtarget Tr_meulage_bavure_204 := [[86.3302578125,-33.0574453125,94.883359375],[0.50240511156018,-0.49002871249699,-0.497396265653287,0.50995874315567],[0,0,0,0],[8.999999E+09,8.999999E+09,8.999999E+09,8.999999E+09,8.999999E+09,8.999999E+09]];
    LOCAL CONST Robtarget Tr_meulage_bavure_205 := [[86.3253203125,-22.593630859375,93.654140625],[0.503524899286381,-0.490358581977652,-0.4962896740168,0.509615243437443],[0,0,0,0],[8.999999E+09,8.999999E+09,8.999999E+09,8.999999E+09,8.999999E+09,8.999999E+09]];
    LOCAL CONST Robtarget Tr_meulage_bavure_206 := [[86.434296875,-18.85490625,93.2149453125],[0.504636525421653,-0.490658646328654,-0.495189770371434,0.509296732085314],[0,0,0,0],[8.999999E+09,8.999999E+09,8.999999E+09,8.999999E+09,8.999999E+09,8.999999E+09]];
    LOCAL CONST Robtarget Tr_meulage_bavure_207 := [[86.44265625,-17.433921875,93.048015625],[0.505642038675138,-0.490831693503953,-0.49419103179346,0.509102741567365],[0,0,0,0],[8.999999E+09,8.999999E+09,8.999999E+09,8.999999E+09,8.999999E+09,8.999999E+09]];
    LOCAL CONST Robtarget Tr_meulage_bavure_208 := [[86.4267890625,-14.44834765625,92.6972890625],[0.506452561017489,-0.490794569861028,-0.493379514660815,0.509119974217093],[0,0,0,0],[8.999999E+09,8.999999E+09,8.999999E+09,8.999999E+09,8.999999E+09,8.999999E+09]];
    LOCAL CONST Robtarget Tr_meulage_bavure_209 := [[86.5483125,-10.74562890625,92.2623203125],[0.507009652181912,-0.490491154057295,-0.492811407411933,0.509408045785095],[0,0,0,0],[8.999999E+09,8.999999E+09,8.999999E+09,8.999999E+09,8.999999E+09,8.999999E+09]];
    LOCAL CONST Robtarget Tr_meulage_bavure_210 := [[86.6441640625,-6.97519921875,91.8193984375],[0.507288681038177,-0.489899326215803,-0.492509451766881,0.5099914550109],[0,0,0,0],[8.999999E+09,8.999999E+09,8.999999E+09,8.999999E+09,8.999999E+09,8.999999E+09]];
    LOCAL CONST Robtarget Tr_meulage_bavure_211 := [[86.7646484375,-1.59844458007813,91.1877734375],[0.507302046994587,-0.489030468248667,-0.492459673973791,0.510859377665928],[0,0,0,0],[8.999999E+09,8.999999E+09,8.999999E+09,8.999999E+09,8.999999E+09,8.999999E+09]];
    LOCAL CONST Robtarget Tr_meulage_bavure_212 := [[86.75403125,0.847050170898437,90.9004921875],[0.507100015686869,-0.487932537445571,-0.492611223203828,0.511962494491473],[0,0,0,0],[8.999999E+09,8.999999E+09,8.999999E+09,8.999999E+09,8.999999E+09,8.999999E+09]];
    LOCAL CONST Robtarget Tr_meulage_bavure_213 := [[86.6206640625,5.52493603515625,90.35096875],[0.506758325739697,-0.486680490410067,-0.492889351008217,0.513223330734695],[0,0,0,0],[8.999999E+09,8.999999E+09,8.999999E+09,8.999999E+09,8.999999E+09,8.999999E+09]];
    LOCAL CONST Robtarget Tr_meulage_bavure_214 := [[86.6286015625,6.52889697265625,90.23303125],[0.50636501941569,-0.485364409287441,-0.493209018329447,0.514549046785343],[0,0,0,0],[8.999999E+09,8.999999E+09,8.999999E+09,8.999999E+09,8.999999E+09,8.999999E+09]];
    LOCAL CONST Robtarget Tr_meulage_bavure_215 := [[86.716125,7.354306640625,90.1360703125],[0.506021936986899,-0.484075711482886,-0.4934732742574,0.515845550949162],[0,0,0,0],[8.999999E+09,8.999999E+09,8.999999E+09,8.999999E+09,8.999999E+09,8.999999E+09]];
    LOCAL CONST Robtarget Tr_meulage_bavure_216 := [[86.4696328125,16.80333984375,89.0260625],[0.505815474777885,-0.482900852897007,-0.493602141890095,0.517024561571378],[0,0,0,0],[8.999999E+09,8.999999E+09,8.999999E+09,8.999999E+09,8.999999E+09,8.999999E+09]];
    LOCAL CONST Robtarget Tr_meulage_bavure_217 := [[86.4443671875,17.54751953125,88.938640625],[0.505809850139581,-0.481899899328049,-0.493537432915405,0.518024791723971],[0,0,0,0],[8.999999E+09,8.999999E+09,8.999999E+09,8.999999E+09,8.999999E+09,8.999999E+09]];
    LOCAL CONST Robtarget Tr_meulage_bavure_218 := [[86.4371328125,18.23687109375,88.85765625],[0.506055635377881,-0.481120927833326,-0.493234374027946,0.518796876417302],[0,0,0,0],[8.999999E+09,8.999999E+09,8.999999E+09,8.999999E+09,8.999999E+09,8.999999E+09]];
    LOCAL CONST Robtarget Tr_meulage_bavure_219 := [[86.2521953125,25.02897265625,88.0597734375],[0.506561034059352,-0.480569555062016,-0.492687334596366,0.519334200538097],[0,0,0,0],[8.999999E+09,8.999999E+09,8.999999E+09,8.999999E+09,8.999999E+09,8.999999E+09]];
    LOCAL CONST Robtarget Tr_meulage_bavure_220 := [[86.0518203125,27.379509765625,87.7836484375],[0.507307901445374,-0.48022995267106,-0.491914764632691,0.519651565979558],[0,0,0,0],[8.999999E+09,8.999999E+09,8.999999E+09,8.999999E+09,8.999999E+09,8.999999E+09]];
    LOCAL CONST Robtarget Tr_meulage_bavure_221 := [[85.996859375,31.103232421875,87.3462109375],[0.508260806274948,-0.48006325002738,-0.490949897850039,0.519786904970609],[0,0,0,0],[8.999999E+09,8.999999E+09,8.999999E+09,8.999999E+09,8.999999E+09,8.999999E+09]];
    LOCAL CONST Robtarget Tr_meulage_bavure_222 := [[85.830140625,33.11876171875,87.1094375],[0.50933182483175,-0.479989452306774,-0.489874574712248,0.519821237482942],[0,0,0,0],[8.999999E+09,8.999999E+09,8.999999E+09,8.999999E+09,8.999999E+09,8.999999E+09]];
    LOCAL CONST Robtarget Tr_meulage_bavure_223 := [[85.7946796875,34.63709765625,86.931078125],[0.510421289602581,-0.47991620793287,-0.488781053779592,0.519849614744384],[0,0,0,0],[8.999999E+09,8.999999E+09,8.999999E+09,8.999999E+09,8.999999E+09,8.999999E+09]];
    LOCAL CONST Robtarget Tr_meulage_bavure_224 := [[85.7939453125,37.69601953125,86.571734375],[0.511387632015262,-0.479709207636207,-0.487799857707369,0.520012562109356],[0,0,0,0],[8.999999E+09,8.999999E+09,8.999999E+09,8.999999E+09,8.999999E+09,8.999999E+09]];
    LOCAL CONST Robtarget Tr_meulage_bavure_225 := [[85.8785703125,43.22671484375,85.92203125],[0.512080090245506,-0.479225370346959,-0.487069325966123,0.520461811560542],[0,0,0,0],[8.999999E+09,8.999999E+09,8.999999E+09,8.999999E+09,8.999999E+09,8.999999E+09]];
    LOCAL CONST Robtarget Tr_meulage_bavure_226 := [[85.818265625,46.49253125,85.5383828125],[0.512304427292084,-0.478292359212782,-0.486766804267496,0.521381502509256],[0,0,0,0],[8.999999E+09,8.999999E+09,8.999999E+09,8.999999E+09,8.999999E+09,8.999999E+09]];
    LOCAL CONST Robtarget Tr_meulage_bavure_227 := [[85.79171875,49.59758203125,85.173625],[0.511808038084647,-0.476681193587554,-0.487118022550624,0.523013961513705],[0,0,0,0],[8.999999E+09,8.999999E+09,8.999999E+09,8.999999E+09,8.999999E+09,8.999999E+09]];
    LOCAL CONST Robtarget Tr_meulage_bavure_228 := [[85.757015625,56.3792890625,84.376953125],[0.510310771370111,-0.474135026613408,-0.488362787217713,0.525624087369379],[0,0,0,0],[8.999999E+09,8.999999E+09,8.999999E+09,8.999999E+09,8.999999E+09,8.999999E+09]];
    LOCAL CONST Robtarget Tr_meulage_bavure_229 := [[85.7904375,60.828609375,83.85428125],[0.507444690826793,-0.47031865818964,-0.490800018592128,0.529542809657881],[0,0,0,0],[8.999999E+09,8.999999E+09,8.999999E+09,8.999999E+09,8.999999E+09,8.999999E+09]];
    LOCAL CONST Robtarget Tr_meulage_bavure_230 := [[85.70428125,69.3919140625,82.8483203125],[0.502783564826386,-0.464851389480305,-0.494744801923186,0.535116299143176],[0,0,0,0],[8.999999E+09,8.999999E+09,8.999999E+09,8.999999E+09,8.999999E+09,8.999999E+09]];
    LOCAL CONST Robtarget Tr_meulage_bavure_231 := [[85.6923203125,69.6727890625,82.815328125],[0.495826739705595,-0.457286398776168,-0.500518618863679,0.542702594298238],[0,0,0,0],[8.999999E+09,8.999999E+09,8.999999E+09,8.999999E+09,8.999999E+09,8.999999E+09]];
    LOCAL CONST Robtarget Tr_meulage_bavure_232 := [[85.6911953125,70.15965625,82.7581328125],[0.485986968057435,-0.447094401897387,-0.508426030260794,0.552653810647869],[0,0,0,0],[8.999999E+09,8.999999E+09,8.999999E+09,8.999999E+09,8.999999E+09,8.999999E+09]];
    LOCAL CONST Robtarget Tr_meulage_bavure_233 := [[85.6990390625,70.79584375,82.6833984375],[0.47262086201403,-0.433715684652381,-0.518694422355538,0.565222364997074],[0,0,0,0],[8.999999E+09,8.999999E+09,8.999999E+09,8.999999E+09,8.999999E+09,8.999999E+09]];
    LOCAL CONST Robtarget Tr_meulage_bavure_234 := [[85.7366953125,77.630734375,81.880484375],[0.455071437034857,-0.416567336059,-0.531397505707381,0.580515574857137],[0,0,0,0],[8.999999E+09,8.999999E+09,8.999999E+09,8.999999E+09,8.999999E+09,8.999999E+09]];
    LOCAL CONST Robtarget Tr_meulage_bavure_235 := [[85.858859375,79.91678125,81.6119375],[0.43271383196824,-0.395114013556226,-0.546405134162145,0.59840211001976],[0,0,0,0],[8.999999E+09,8.999999E+09,8.999999E+09,8.999999E+09,8.999999E+09,8.999999E+09]];
    LOCAL CONST Robtarget Tr_meulage_bavure_236 := [[85.9930078125,84.9015703125,81.026359375],[0.405118760110084,-0.368992295386907,-0.563274162889688,0.618421938140046],[0,0,0,0],[8.999999E+09,8.999999E+09,8.999999E+09,8.999999E+09,8.999999E+09,8.999999E+09]];
    LOCAL CONST Robtarget Tr_meulage_bavure_237 := [[85.841640625,85.8825625,80.9111171875],[0.372233894058798,-0.33819906876735,-0.581226229709356,0.639718209758459],[0,0,0,0],[8.999999E+09,8.999999E+09,8.999999E+09,8.999999E+09,8.999999E+09,8.999999E+09]];
    LOCAL CONST Robtarget Tr_meulage_bavure_238 := [[85.4545625,88.4115234375,80.61403125],[0.334607175724312,-0.30325897253494,-0.599171915071483,0.661108954500257],[0,0,0,0],[8.999999E+09,8.999999E+09,8.999999E+09,8.999999E+09,8.999999E+09,8.999999E+09]];
    LOCAL CONST Robtarget Tr_meulage_bavure_239 := [[85.2495390625,88.7909921875,80.569453125],[0.293519748817148,-0.26536956253418,-0.615904509227877,0.681239156132047],[0,0,0,0],[8.999999E+09,8.999999E+09,8.999999E+09,8.999999E+09,8.999999E+09,8.999999E+09]];
    LOCAL CONST Robtarget Tr_meulage_bavure_240 := [[83.979,90.90378125,80.3212578125],[0.250807295302673,-0.226200440496082,-0.630384335518628,0.698959691881495],[0,0,0,0],[8.999999E+09,8.999999E+09,8.999999E+09,8.999999E+09,8.999999E+09,8.999999E+09]];
    LOCAL CONST Robtarget Tr_meulage_bavure_241 := [[82.4261796875,92.0024609375,80.1921953125],[0.208565091223179,-0.187649972088293,-0.64198666785841,0.713541315545488],[0,0,0,0],[8.999999E+09,8.999999E+09,8.999999E+09,8.999999E+09,8.999999E+09,8.999999E+09]];
    LOCAL CONST Robtarget Tr_meulage_bavure_242 := [[80.9743984375,92.9609921875,80.07959375],[0.168720140808233,-0.151439202480963,-0.650574293021987,0.724812231751453],[0,0,0,0],[8.999999E+09,8.999999E+09,8.999999E+09,8.999999E+09,8.999999E+09,8.999999E+09]];
    LOCAL CONST Robtarget Tr_meulage_bavure_243 := [[78.73303125,93.380953125,80.0302578125],[0.132682930232438,-0.118813598636844,-0.656432270646719,0.733058826328072],[0,0,0,0],[8.999999E+09,8.999999E+09,8.999999E+09,8.999999E+09,8.999999E+09,8.999999E+09]];
    LOCAL CONST Robtarget Tr_meulage_bavure_244 := [[77.1343046875,93.63525,80.0003828125],[0.101302877005038,-0.0905034401421771,-0.660063019124753,0.738825869347338],[0,0,0,0],[8.999999E+09,8.999999E+09,8.999999E+09,8.999999E+09,8.999999E+09,8.999999E+09]];
    LOCAL CONST Robtarget Tr_meulage_bavure_245 := [[76.800078125,93.6117265625,80.0031484375],[0.074875339051969,-0.0667409577332813,-0.662038478573092,0.742727662775073],[0,0,0,0],[8.999999E+09,8.999999E+09,8.999999E+09,8.999999E+09,8.999999E+09,8.999999E+09]];
    LOCAL CONST Robtarget Tr_meulage_bavure_246 := [[72.9012734375,93.4064453125,80.027265625],[0.0532990236288366,-0.0474030099449921,-0.662875457886105,0.745324289192735],[0,0,0,0],[8.999999E+09,8.999999E+09,8.999999E+09,8.999999E+09,8.999999E+09,8.999999E+09]];
    LOCAL CONST Robtarget Tr_meulage_bavure_247 := [[66.3278828125,92.819234375,80.0962421875],[0.0362156982171738,-0.0321394640625369,-0.662982057246187,0.747067781276927],[0,0,0,0],[8.999999E+09,8.999999E+09,8.999999E+09,8.999999E+09,8.999999E+09,8.999999E+09]];
    LOCAL CONST Robtarget Tr_meulage_bavure_248 := [[63.35751171875,92.6392890625,80.1173828125],[0.0231325701371251,-0.0204852970313237,-0.662654280298693,0.748287739847588],[0,0,0,0],[8.999999E+09,8.999999E+09,8.999999E+09,8.999999E+09,8.999999E+09,8.999999E+09]];
    LOCAL CONST Robtarget Tr_meulage_bavure_249 := [[54.66980078125,92.5391171875,80.1291484375],[0.0134853222170677,-0.01191737762901,-0.662094175016074,0.749204528553408],[0,0,0,0],[8.999999E+09,8.999999E+09,8.999999E+09,8.999999E+09,8.999999E+09,8.999999E+09]];
    LOCAL CONST Robtarget Tr_meulage_bavure_250 := [[50.84353515625,92.4651953125,80.1378359375],[0.00670173422219705,-0.00591063549651315,-0.661427877617114,0.749955541253855],[0,0,0,0],[8.999999E+09,8.999999E+09,8.999999E+09,8.999999E+09,8.999999E+09,8.999999E+09]];
    LOCAL CONST Robtarget Tr_meulage_bavure_251 := [[45.43997265625,92.34771875,80.151640625],[0.00219554039993453,-0.00193260299222823,-0.660726687977192,0.75062086864323],[0,0,0,0],[8.999999E+09,8.999999E+09,8.999999E+09,8.999999E+09,8.999999E+09,8.999999E+09]];
    LOCAL CONST Robtarget Tr_meulage_bavure_252 := [[32.35153125,92.2526328125,80.1628046875],[0.000565530709692145,-0.000496867348034901,0.660028830734829,-0.751239892375711],[0,0,0,0],[8.999999E+09,8.999999E+09,8.999999E+09,8.999999E+09,8.999999E+09,8.999999E+09]];
    LOCAL CONST Robtarget Tr_meulage_bavure_253 := [[22.68276953125,92.266640625,80.1611640625],[0.00202943746266615,-0.00177983240314181,0.659356713422326,-0.751825403963653],[0,0,0,0],[8.999999E+09,8.999999E+09,8.999999E+09,8.999999E+09,8.999999E+09,8.999999E+09]];
    LOCAL CONST Robtarget Tr_meulage_bavure_254 := [[17.4424140625,92.1639453125,80.1732265625],[0.00264288218607428,-0.00231382727348544,0.658710992407752,-0.752387858659543],[0,0,0,0],[8.999999E+09,8.999999E+09,8.999999E+09,8.999999E+09,8.999999E+09,8.999999E+09]];
    LOCAL CONST Robtarget Tr_meulage_bavure_255 := [[16.2614140625,92.1460078125,80.175328125],[0.00276071057108996,-0.00241297962390337,0.65809196448547,-0.7529286302739],[0,0,0,0],[8.999999E+09,8.999999E+09,8.999999E+09,8.999999E+09,8.999999E+09,8.999999E+09]];
    LOCAL CONST Robtarget Tr_meulage_bavure_256 := [[5.9198916015625,91.86640625,80.2081796875],[0.00272449474038209,-0.00237756912704035,0.657502987963104,-0.753443259385234],[0,0,0,0],[8.999999E+09,8.999999E+09,8.999999E+09,8.999999E+09,8.999999E+09,8.999999E+09]];
    LOCAL CONST Robtarget Tr_meulage_bavure_257 := [[2.16122436523438,91.810453125,80.21475],[0.00285977825819117,-0.00249189197577326,0.656943509644324,-0.753930260222319],[0,0,0,0],[8.999999E+09,8.999999E+09,8.999999E+09,8.999999E+09,8.999999E+09,8.999999E+09]];
